LIN {X 0,Y 432.358,Z 386.63,A -85,B 0,C 180,E1 -9401.61,E2 -9401.61} C_VEL
LIN {X 0,Y 432.364,Z 386.63,A -85,B 0,C 180,E1 -9404.344,E2 -9404.344} C_VEL
LIN {X 0,Y 432.353,Z 386.63,A -85,B 0,C 180,E1 -9407.012,E2 -9407.012} C_VEL
LIN {X 0,Y 432.346,Z 386.632,A -85,B 0,C 180,E1 -9409.819,E2 -9409.819} C_VEL
LIN {X 0,Y 432.307,Z 386.637,A -85,B 0,C 180,E1 -9413.026,E2 -9413.026} C_VEL
LIN {X 0,Y 432.344,Z 386.755,A -85,B 0,C 180,E1 -9413.32,E2 -9413.32} C_VEL
LIN {X 0,Y 433.977,Z 394.809,A -85,B 0,C 180,E1 -9416.595,E2 -9416.595} C_VEL
LIN {X 0,Y 435.011,Z 400.873,A -85,B 0,C 180,E1 -9418.9,E2 -9418.9} C_VEL
LIN {X 0,Y 434.635,Z 406.92,A -85,B 0,C 180,E1 -9420.984,E2 -9420.984} C_VEL
LIN {X 0,Y 433.713,Z 417.772,A -85,B 0,C 180,E1 -9424.573,E2 -9424.573} C_VEL
LIN {X 0,Y 432.959,Z 428.81,A -85,B 0,C 180,E1 -9428.081,E2 -9428.081} C_VEL
LIN {X 0,Y 432.347,Z 440.008,A -85,B 0,C 180,E1 -9431.522,E2 -9431.522} C_VEL
LIN {X 0,Y 432.076,Z 446.933,A -85,B 0,C 180,E1 -9433.599,E2 -9433.599} C_VEL
LIN {X 0,Y 434.037,Z 460.55,A -85,B 0,C 180,E1 -9434.04,E2 -9434.04} C_VEL
LIN {X 0,Y 435.084,Z 471.816,A -85,B 0,C 180,E1 -9434.545,E2 -9434.545} C_VEL
LIN {X 0,Y 434.478,Z 484.277,A -85,B 0,C 180,E1 -9435.243,E2 -9435.243} C_VEL
LIN {X 0,Y 433.851,Z 495.5,A -85,B 0,C 180,E1 -9436.066,E2 -9436.066} C_VEL
LIN {X 0,Y 433.278,Z 505.592,A -85,B 0,C 180,E1 -9436.996,E2 -9436.996} C_VEL
LIN {X 0,Y 432.825,Z 514.915,A -85,B 0,C 180,E1 -9438.054,E2 -9438.054} C_VEL
LIN {X 0,Y 432.276,Z 523.539,A -85,B 0,C 180,E1 -9439.226,E2 -9439.226} C_VEL
LIN {X 0,Y 431.847,Z 531.941,A -85,B 0,C 180,E1 -9440.636,E2 -9440.636} C_VEL
LIN {X 0,Y 431.545,Z 538.678,A -85,B 0,C 180,E1 -9442.045,E2 -9442.045} C_VEL
LIN {X 0,Y 431.34,Z 544.033,A -85,B 0,C 180,E1 -9443.453,E2 -9443.453} C_VEL
LIN {X 0,Y 431.31,Z 548.179,A -85,B 0,C 180,E1 -9444.86,E2 -9444.86} C_VEL
LIN {X 0,Y 431.221,Z 551.229,A -85,B 0,C 180,E1 -9446.264,E2 -9446.264} C_VEL
LIN {X 0,Y 431.268,Z 552.713,A -85,B 0,C 180,E1 -9447.2,E2 -9447.2} C_VEL
LIN {X 0,Y 431.273,Z 553.741,A -85,B 0,C 180,E1 -9448.134,E2 -9448.134} C_VEL
LIN {X 0,Y 431.222,Z 554.368,A -85,B 0,C 180,E1 -9449.068,E2 -9449.068} C_VEL
LIN {X 0,Y 431.193,Z 554.599,A -85,B 0,C 180,E1 -9450.002,E2 -9450.002} C_VEL
LIN {X 0,Y 431.223,Z 554.385,A -85,B 0,C 180,E1 -9450.936,E2 -9450.936} C_VEL
LIN {X 0,Y 431.285,Z 553.758,A -85,B 0,C 180,E1 -9451.87,E2 -9451.87} C_VEL
LIN {X 0,Y 431.269,Z 552.732,A -85,B 0,C 180,E1 -9452.804,E2 -9452.804} C_VEL
LIN {X 0,Y 431.223,Z 551.283,A -85,B 0,C 180,E1 -9453.74,E2 -9453.74} C_VEL
LIN {X 0,Y 431.313,Z 548.261,A -85,B 0,C 180,E1 -9455.144,E2 -9455.144} C_VEL
LIN {X 0,Y 431.379,Z 544.16,A -85,B 0,C 180,E1 -9456.55,E2 -9456.55} C_VEL
LIN {X 0,Y 431.599,Z 537.834,A -85,B 0,C 180,E1 -9458.193,E2 -9458.193} C_VEL
LIN {X 0,Y 431.932,Z 530.939,A -85,B 0,C 180,E1 -9459.602,E2 -9459.602} C_VEL
LIN {X 0,Y 432.371,Z 522.327,A -85,B 0,C 180,E1 -9461.012,E2 -9461.012} C_VEL
LIN {X 0,Y 432.952,Z 513.464,A -85,B 0,C 180,E1 -9462.184,E2 -9462.184} C_VEL
LIN {X 0,Y 433.444,Z 503.391,A -85,B 0,C 180,E1 -9463.278,E2 -9463.278} C_VEL
LIN {X 0,Y 434.074,Z 493.107,A -85,B 0,C 180,E1 -9464.177,E2 -9464.177} C_VEL
LIN {X 0,Y 434.75,Z 481.287,A -85,B 0,C 180,E1 -9464.992,E2 -9464.992} C_VEL
LIN {X 0,Y 435.121,Z 470.397,A -85,B 0,C 180,E1 -9465.578,E2 -9465.578} C_VEL
LIN {X 0,Y 433.729,Z 457.18,A -85,B 0,C 180,E1 -9466.168,E2 -9466.168} C_VEL
LIN {X 0,Y 432.074,Z 446.577,A -85,B 0,C 180,E1 -9466.534,E2 -9466.534} C_VEL
LIN {X 0,Y 432.581,Z 435.274,A -85,B 0,C 180,E1 -9469.95,E2 -9469.95} C_VEL
LIN {X 0,Y 433.125,Z 425.632,A -85,B 0,C 180,E1 -9472.921,E2 -9472.921} C_VEL
LIN {X 0,Y 433.821,Z 416.066,A -85,B 0,C 180,E1 -9475.94,E2 -9475.94} C_VEL
LIN {X 0,Y 434.748,Z 404.887,A -85,B 0,C 180,E1 -9479.566,E2 -9479.566} C_VEL
LIN {X 0,Y 434.881,Z 400.204,A -85,B 0,C 180,E1 -9481.142,E2 -9481.142} C_VEL
LIN {X 0,Y 433.401,Z 391.79,A -85,B 0,C 180,E1 -9484.206,E2 -9484.206} C_VEL
LIN {X 0,Y 432.35,Z 386.632,A -85,B 0,C 180,E1 -9486.25,E2 -9486.25} C_VEL
LIN {X 0,Y 432.309,Z 386.636,A -85,B 0,C 180,E1 -9489.349,E2 -9489.349} C_VEL
LIN {X 0,Y 432.309,Z 386.637,A -85,B 0,C 180,E1 -9491.802,E2 -9491.802} C_VEL
LIN {X 0,Y 432.338,Z 386.63,A -85,B 0,C 180,E1 -9494.348,E2 -9494.348} C_VEL
LIN {X 0,Y 432.31,Z 386.633,A -85,B 0,C 180,E1 -9497.019,E2 -9497.019} C_VEL
LIN {X 0,Y 432.296,Z 386.633,A -85,B 0,C 180,E1 -9499.828,E2 -9499.828} C_VEL
LIN {X 0,Y 432.313,Z 386.634,A -85,B 0,C 180,E1 -9503.022,E2 -9503.022} C_VEL
LIN {X 0,Y 432.339,Z 386.632,A -85,B 0,C 180,E1 -9506.002,E2 -9506.002} C_VEL
LIN {X 0,Y 432.35,Z 386.631,A -85,B 0,C 180,E1 -9509.491,E2 -9509.491} C_VEL
LIN {X 0,Y 432.323,Z 386.634,A -85,B 0,C 180,E1 -9511.872,E2 -9511.872} C_VEL
LIN {X 0,Y 432.353,Z 386.629,A -85,B 0,C 180,E1 -9515.548,E2 -9515.548} C_VEL
LIN {X 0,Y 432.356,Z 386.63,A -85,B 0,C 180,E1 -9519.046,E2 -9519.046} C_VEL
LIN {X 0,Y 432.383,Z 386.628,A -85,B 0,C 180,E1 -9522.011,E2 -9522.011} C_VEL
LIN {X 0,Y 432.4,Z 386.625,A -85,B 0,C 180,E1 -9524.926,E2 -9524.926} C_VEL
LIN {X 0,Y 432.464,Z 386.618,A -85,B 0,C 180,E1 -9527.803,E2 -9527.803} C_VEL
LIN {X 0,Y 432.452,Z 386.619,A -85,B 0,C 180,E1 -9531.589,E2 -9531.589} C_VEL
LIN {X 0,Y 432.557,Z 386.607,A -85,B 0,C 180,E1 -9534.405,E2 -9534.405} C_VEL
LIN {X 0,Y 432.238,Z 386.721,A -85,B 0,C 180,E1 -9536.154,E2 -9536.154} C_VEL
LIN {X 0,Y 432.548,Z 392.214,A -85,B 0,C 180,E1 -9538.603,E2 -9538.603} C_VEL
LIN {X 0,Y 432.354,Z 397.392,A -85,B 0,C 180,E1 -9540.931,E2 -9540.931} C_VEL
LIN {X 0,Y 432.129,Z 406.596,A -85,B 0,C 180,E1 -9545.132,E2 -9545.132} C_VEL
LIN {X 0,Y 432.005,Z 412.681,A -85,B 0,C 180,E1 -9547.948,E2 -9547.948} C_VEL
LIN {X 0,Y 431.852,Z 419.741,A -85,B 0,C 180,E1 -9551.261,E2 -9551.261} C_VEL
LIN {X 0,Y 431.713,Z 426.157,A -85,B 0,C 180,E1 -9554.284,E2 -9554.284} C_VEL
LIN {X 0,Y 434.813,Z 440.469,A -85,B 0,C 180,E1 -9554.898,E2 -9554.898} C_VEL
LIN {X 0,Y 435.966,Z 447.264,A -85,B 0,C 180,E1 -9555.246,E2 -9555.246} C_VEL
LIN {X 0,Y 435.35,Z 459.685,A -85,B 0,C 180,E1 -9555.928,E2 -9555.928} C_VEL
LIN {X 0,Y 434.713,Z 471.741,A -85,B 0,C 180,E1 -9556.797,E2 -9556.797} C_VEL
LIN {X 0,Y 434.084,Z 482.032,A -85,B 0,C 180,E1 -9557.739,E2 -9557.739} C_VEL
LIN {X 0,Y 433.389,Z 492.493,A -85,B 0,C 180,E1 -9558.925,E2 -9558.925} C_VEL
LIN {X 0,Y 432.83,Z 501.477,A -85,B 0,C 180,E1 -9560.184,E2 -9560.184} C_VEL
LIN {X 0,Y 432.238,Z 510.153,A -85,B 0,C 180,E1 -9561.709,E2 -9561.709} C_VEL
LIN {X 0,Y 431.798,Z 517.081,A -85,B 0,C 180,E1 -9563.247,E2 -9563.247} C_VEL
LIN {X 0,Y 431.546,Z 521.85,A -85,B 0,C 180,E1 -9564.594,E2 -9564.594} C_VEL
LIN {X 0,Y 431.353,Z 526.477,A -85,B 0,C 180,E1 -9566.347,E2 -9566.347} C_VEL
LIN {X 0,Y 431.25,Z 528.08,A -85,B 0,C 180,E1 -9567.149,E2 -9567.149} C_VEL
LIN {X 0,Y 431.151,Z 529.853,A -85,B 0,C 180,E1 -9568.328,E2 -9568.328} C_VEL
LIN {X 0,Y 431.08,Z 530.807,A -85,B 0,C 180,E1 -9569.281,E2 -9569.281} C_VEL
LIN {X 0,Y 431.042,Z 531.392,A -85,B 0,C 180,E1 -9570.361,E2 -9570.361} C_VEL
LIN {X 0,Y 431.038,Z 531.205,A -85,B 0,C 180,E1 -9572.02,E2 -9572.02} C_VEL
LIN {X 0,Y 431.105,Z 529.669,A -85,B 0,C 180,E1 -9573.754,E2 -9573.754} C_VEL
LIN {X 0,Y 431.252,Z 526.839,A -85,B 0,C 180,E1 -9575.427,E2 -9575.427} C_VEL
LIN {X 0,Y 431.486,Z 522.666,A -85,B 0,C 180,E1 -9577.06,E2 -9577.06} C_VEL
LIN {X 0,Y 431.725,Z 517.333,A -85,B 0,C 180,E1 -9578.611,E2 -9578.611} C_VEL
LIN {X 0,Y 432.081,Z 510.568,A -85,B 0,C 180,E1 -9580.138,E2 -9580.138} C_VEL
LIN {X 0,Y 432.607,Z 502.081,A -85,B 0,C 180,E1 -9581.641,E2 -9581.641} C_VEL
LIN {X 0,Y 433.113,Z 494.004,A -85,B 0,C 180,E1 -9582.804,E2 -9582.804} C_VEL
LIN {X 0,Y 433.662,Z 485.008,A -85,B 0,C 180,E1 -9583.876,E2 -9583.876} C_VEL
LIN {X 0,Y 434.24,Z 474.608,A -85,B 0,C 180,E1 -9584.884,E2 -9584.884} C_VEL
LIN {X 0,Y 434.859,Z 463.18,A -85,B 0,C 180,E1 -9585.769,E2 -9585.769} C_VEL
LIN {X 0,Y 435.514,Z 450.906,A -85,B 0,C 180,E1 -9586.502,E2 -9586.502} C_VEL
LIN {X 0,Y 435.473,Z 445.507,A -85,B 0,C 180,E1 -9586.771,E2 -9586.771} C_VEL
LIN {X 0,Y 433.078,Z 432.684,A -85,B 0,C 180,E1 -9587.349,E2 -9587.349} C_VEL
LIN {X 0,Y 431.639,Z 425.615,A -85,B 0,C 180,E1 -9587.608,E2 -9587.608} C_VEL
LIN {X 0,Y 431.733,Z 419.417,A -85,B 0,C 180,E1 -9590.589,E2 -9590.589} C_VEL
LIN {X 0,Y 431.88,Z 412.017,A -85,B 0,C 180,E1 -9594.137,E2 -9594.137} C_VEL
LIN {X 0,Y 432.033,Z 406.117,A -85,B 0,C 180,E1 -9596.977,E2 -9596.977} C_VEL
LIN {X 0,Y 432.172,Z 399.276,A -85,B 0,C 180,E1 -9600.263,E2 -9600.263} C_VEL
LIN {X 0,Y 432.252,Z 392.712,A -85,B 0,C 180,E1 -9603.411,E2 -9603.411} C_VEL
LIN {X 0,Y 432.451,Z 386.619,A -85,B 0,C 180,E1 -9606.408,E2 -9606.408} C_VEL
LIN {X 0,Y 432.34,Z 386.632,A -85,B 0,C 180,E1 -9610.038,E2 -9610.038} C_VEL
LIN {X 0,Y 432.414,Z 386.624,A -85,B 0,C 180,E1 -9613.52,E2 -9613.52} C_VEL
LIN {X 0,Y 432.432,Z 386.62,A -85,B 0,C 180,E1 -9617.195,E2 -9617.195} C_VEL
LIN {X 0,Y 432.442,Z 386.618,A -85,B 0,C 180,E1 -9620.645,E2 -9620.645} C_VEL
LIN {X 0,Y 432.512,Z 386.61,A -85,B 0,C 180,E1 -9622.409,E2 -9622.409} C_VEL
LIN {X 0,Y 431.783,Z 386.704,A -85,B 0,C 180,E1 -9623.186,E2 -9623.186} C_VEL
LIN {X 0,Y 428.797,Z 387.08,A -85,B 0,C 180,E1 -9624.447,E2 -9624.447} C_VEL
LIN {X 0,Y 426.351,Z 387.384,A -85,B 0,C 180,E1 -9625.465,E2 -9625.465} C_VEL
LIN {X 0,Y 425.387,Z 387.502,A -85,B 0,C 180,E1 -9626.253,E2 -9626.253} C_VEL
LIN {X 0,Y 425.354,Z 387.503,A -85,B 0,C 180,E1 -9626.519,E2 -9626.519} C_VEL
LIN {X 0,Y 425.564,Z 387.52,A -85,B 0,C 180,E1 -9629.17,E2 -9629.17} C_VEL
LIN {X 0,Y 425.818,Z 388.833,A -85,B 0,C 180,E1 -9629.998,E2 -9629.998} C_VEL
LIN {X 0,Y 425.455,Z 393.602,A -85,B 0,C 180,E1 -9632.838,E2 -9632.838} C_VEL
LIN {X 0,Y 425.307,Z 398.421,A -85,B 0,C 180,E1 -9635.688,E2 -9635.688} C_VEL
LIN {X 0,Y 425.074,Z 403.376,A -85,B 0,C 180,E1 -9638.555,E2 -9638.555} C_VEL
LIN {X 0,Y 424.886,Z 410.151,A -85,B 0,C 180,E1 -9642.415,E2 -9642.415} C_VEL
LIN {X 0,Y 424.587,Z 417.168,A -85,B 0,C 180,E1 -9646.341,E2 -9646.341} C_VEL
LIN {X 0,Y 424.462,Z 422.693,A -85,B 0,C 180,E1 -9649.392,E2 -9649.392} C_VEL
LIN {X 0,Y 426.781,Z 435.095,A -85,B 0,C 180,E1 -9649.953,E2 -9649.953} C_VEL
LIN {X 0,Y 427.572,Z 441.78,A -85,B 0,C 180,E1 -9650.328,E2 -9650.328} C_VEL
LIN {X 0,Y 427.066,Z 453.282,A -85,B 0,C 180,E1 -9651.096,E2 -9651.096} C_VEL
LIN {X 0,Y 426.546,Z 462.376,A -85,B 0,C 180,E1 -9651.884,E2 -9651.884} C_VEL
LIN {X 0,Y 426.089,Z 471.591,A -85,B 0,C 180,E1 -9652.9,E2 -9652.9} C_VEL
LIN {X 0,Y 425.551,Z 480.362,A -85,B 0,C 180,E1 -9654.123,E2 -9654.123} C_VEL
LIN {X 0,Y 425.108,Z 487.845,A -85,B 0,C 180,E1 -9655.454,E2 -9655.454} C_VEL
LIN {X 0,Y 424.771,Z 493.266,A -85,B 0,C 180,E1 -9656.691,E2 -9656.691} C_VEL
LIN {X 0,Y 424.515,Z 498.155,A -85,B 0,C 180,E1 -9658.136,E2 -9658.136} C_VEL
LIN {X 0,Y 424.323,Z 502.024,A -85,B 0,C 180,E1 -9659.791,E2 -9659.791} C_VEL
LIN {X 0,Y 424.173,Z 503.721,A -85,B 0,C 180,E1 -9660.903,E2 -9660.903} C_VEL
LIN {X 0,Y 424.093,Z 504.894,A -85,B 0,C 180,E1 -9662.311,E2 -9662.311} C_VEL
LIN {X 0,Y 424.088,Z 505.08,A -85,B 0,C 180,E1 -9663.15,E2 -9663.15} C_VEL
LIN {X 0,Y 424.152,Z 504.719,A -85,B 0,C 180,E1 -9664.285,E2 -9664.285} C_VEL
LIN {X 0,Y 424.288,Z 503.202,A -85,B 0,C 180,E1 -9665.743,E2 -9665.743} C_VEL
LIN {X 0,Y 424.497,Z 500.104,A -85,B 0,C 180,E1 -9667.374,E2 -9667.374} C_VEL
LIN {X 0,Y 424.813,Z 495.456,A -85,B 0,C 180,E1 -9668.963,E2 -9668.963} C_VEL
LIN {X 0,Y 425.089,Z 490.857,A -85,B 0,C 180,E1 -9670.146,E2 -9670.146} C_VEL
LIN {X 0,Y 425.417,Z 484.917,A -85,B 0,C 180,E1 -9671.358,E2 -9671.358} C_VEL
LIN {X 0,Y 425.862,Z 477.403,A -85,B 0,C 180,E1 -9672.576,E2 -9672.576} C_VEL
LIN {X 0,Y 426.409,Z 469.473,A -85,B 0,C 180,E1 -9673.605,E2 -9673.605} C_VEL
LIN {X 0,Y 426.951,Z 460.386,A -85,B 0,C 180,E1 -9674.547,E2 -9674.547} C_VEL
LIN {X 0,Y 427.53,Z 450.085,A -85,B 0,C 180,E1 -9675.385,E2 -9675.385} C_VEL
LIN {X 0,Y 427.88,Z 440.687,A -85,B 0,C 180,E1 -9675.974,E2 -9675.974} C_VEL
LIN {X 0,Y 425.844,Z 429.204,A -85,B 0,C 180,E1 -9676.594,E2 -9676.594} C_VEL
LIN {X 0,Y 424.545,Z 423.172,A -85,B 0,C 180,E1 -9676.876,E2 -9676.876} C_VEL
LIN {X 0,Y 424.685,Z 416.884,A -85,B 0,C 180,E1 -9680.423,E2 -9680.423} C_VEL
LIN {X 0,Y 424.889,Z 410.362,A -85,B 0,C 180,E1 -9684.139,E2 -9684.139} C_VEL
LIN {X 0,Y 425.09,Z 404.684,A -85,B 0,C 180,E1 -9687.471,E2 -9687.471} C_VEL
LIN {X 0,Y 425.306,Z 399.882,A -85,B 0,C 180,E1 -9690.282,E2 -9690.282} C_VEL
LIN {X 0,Y 425.57,Z 394.467,A -85,B 0,C 180,E1 -9693.52,E2 -9693.52} C_VEL
LIN {X 0,Y 425.68,Z 391.017,A -85,B 0,C 180,E1 -9695.623,E2 -9695.623} C_VEL
LIN {X 0,Y 425.345,Z 387.506,A -85,B 0,C 180,E1 -9698.001,E2 -9698.001} C_VEL
LIN {X 0,Y 425.341,Z 387.508,A -85,B 0,C 180,E1 -9700.703,E2 -9700.703} C_VEL
LIN {X 0,Y 425.364,Z 387.505,A -85,B 0,C 180,E1 -9703.688,E2 -9703.688} C_VEL
LIN {X 0,Y 425.41,Z 387.496,A -85,B 0,C 180,E1 -9707.598,E2 -9707.598} C_VEL
LIN {X 0,Y 425.42,Z 387.495,A -85,B 0,C 180,E1 -9711.45,E2 -9711.45} C_VEL
LIN {X 0,Y 425.556,Z 387.478,A -85,B 0,C 180,E1 -9714.314,E2 -9714.314} C_VEL
LIN {X 0,Y 425.554,Z 387.476,A -85,B 0,C 180,E1 -9718.108,E2 -9718.108} C_VEL
LIN {X 0,Y 425.681,Z 387.461,A -85,B 0,C 180,E1 -9720,E2 -9720} C_VEL
LIN {X 0,Y 425.543,Z 387.479,A -85,B 0,C 180,E1 -9722.84,E2 -9722.84} C_VEL
LIN {X 0,Y 425.556,Z 387.478,A -85,B 0,C 180,E1 -9725.687,E2 -9725.687} C_VEL
LIN {X 0,Y 425.42,Z 387.495,A -85,B 0,C 180,E1 -9728.551,E2 -9728.551} C_VEL
LIN {X 0,Y 425.411,Z 387.493,A -85,B 0,C 180,E1 -9732.402,E2 -9732.402} C_VEL
LIN {X 0,Y 425.377,Z 387.497,A -85,B 0,C 180,E1 -9736.313,E2 -9736.313} C_VEL
LIN {X 0,Y 425.341,Z 387.505,A -85,B 0,C 180,E1 -9739.65,E2 -9739.65} C_VEL
LIN {X 0,Y 425.283,Z 387.511,A -85,B 0,C 180,E1 -9742.339,E2 -9742.339} C_VEL
LIN {X 0,Y 425.275,Z 387.511,A -85,B 0,C 180,E1 -9745.447,E2 -9745.447} C_VEL
LIN {X 0,Y 425.318,Z 387.508,A -85,B 0,C 180,E1 -9748.633,E2 -9748.633} C_VEL
LIN {X 0,Y 425.247,Z 387.512,A -85,B 0,C 180,E1 -9751.929,E2 -9751.929} C_VEL
LIN {X 0,Y 425.283,Z 387.512,A -85,B 0,C 180,E1 -9755.338,E2 -9755.338} C_VEL
LIN {X 0,Y 425.297,Z 387.51,A -85,B 0,C 180,E1 -9759.048,E2 -9759.048} C_VEL
LIN {X 0,Y 425.317,Z 387.507,A -85,B 0,C 180,E1 -9762.648,E2 -9762.648} C_VEL
LIN {X 0,Y 425.321,Z 387.508,A -85,B 0,C 180,E1 -9766.056,E2 -9766.056} C_VEL
LIN {X 0,Y 425.297,Z 387.509,A -85,B 0,C 180,E1 -9768.628,E2 -9768.628} C_VEL
LIN {X 0,Y 425.313,Z 387.508,A -85,B 0,C 180,E1 -9771.107,E2 -9771.107} C_VEL
LIN {X 0,Y 425.294,Z 387.61,A -85,B 0,C 180,E1 -9772.907,E2 -9772.907} C_VEL
LIN {X 0,Y 426.79,Z 394.85,A -85,B 0,C 180,E1 -9775.956,E2 -9775.956} C_VEL
LIN {X 0,Y 427.974,Z 401.737,A -85,B 0,C 180,E1 -9778.641,E2 -9778.641} C_VEL
LIN {X 0,Y 427.951,Z 405.329,A -85,B 0,C 180,E1 -9779.945,E2 -9779.945} C_VEL
LIN {X 0,Y 427.036,Z 414.755,A -85,B 0,C 180,E1 -9783.144,E2 -9783.144} C_VEL
LIN {X 0,Y 426.317,Z 423.905,A -85,B 0,C 180,E1 -9786.181,E2 -9786.181} C_VEL
LIN {X 0,Y 425.606,Z 435.019,A -85,B 0,C 180,E1 -9789.713,E2 -9789.713} C_VEL
LIN {X 0,Y 425.052,Z 446.04,A -85,B 0,C 180,E1 -9793.134,E2 -9793.134} C_VEL
LIN {X 0,Y 425.03,Z 446.677,A -85,B 0,C 180,E1 -9793.328,E2 -9793.328} C_VEL
LIN {X 0,Y 427.067,Z 460.804,A -85,B 0,C 180,E1 -9793.803,E2 -9793.803} C_VEL
LIN {X 0,Y 428.185,Z 472.48,A -85,B 0,C 180,E1 -9794.35,E2 -9794.35} C_VEL
LIN {X 0,Y 427.587,Z 483.807,A -85,B 0,C 180,E1 -9794.999,E2 -9794.999} C_VEL
LIN {X 0,Y 426.919,Z 495.116,A -85,B 0,C 180,E1 -9795.84,E2 -9795.84} C_VEL
LIN {X 0,Y 426.331,Z 504.628,A -85,B 0,C 180,E1 -9796.725,E2 -9796.725} C_VEL
LIN {X 0,Y 425.826,Z 514.507,A -85,B 0,C 180,E1 -9797.855,E2 -9797.855} C_VEL
LIN {X 0,Y 425.25,Z 523.184,A -85,B 0,C 180,E1 -9799.046,E2 -9799.046} C_VEL
LIN {X 0,Y 424.793,Z 531.626,A -85,B 0,C 180,E1 -9800.479,E2 -9800.479} C_VEL
LIN {X 0,Y 424.496,Z 538.388,A -85,B 0,C 180,E1 -9801.912,E2 -9801.912} C_VEL
LIN {X 0,Y 424.255,Z 543.764,A -85,B 0,C 180,E1 -9803.343,E2 -9803.343} C_VEL
LIN {X 0,Y 424.221,Z 547.93,A -85,B 0,C 180,E1 -9804.774,E2 -9804.774} C_VEL
LIN {X 0,Y 424.13,Z 550.997,A -85,B 0,C 180,E1 -9806.202,E2 -9806.202} C_VEL
LIN {X 0,Y 424.164,Z 552.497,A -85,B 0,C 180,E1 -9807.153,E2 -9807.153} C_VEL
LIN {X 0,Y 424.194,Z 553.533,A -85,B 0,C 180,E1 -9808.103,E2 -9808.103} C_VEL
LIN {X 0,Y 424.139,Z 554.167,A -85,B 0,C 180,E1 -9809.053,E2 -9809.053} C_VEL
LIN {X 0,Y 424.109,Z 554.405,A -85,B 0,C 180,E1 -9810.002,E2 -9810.002} C_VEL
LIN {X 0,Y 424.141,Z 554.202,A -85,B 0,C 180,E1 -9810.952,E2 -9810.952} C_VEL
LIN {X 0,Y 424.205,Z 553.581,A -85,B 0,C 180,E1 -9811.901,E2 -9811.901} C_VEL
LIN {X 0,Y 424.165,Z 552.557,A -85,B 0,C 180,E1 -9812.851,E2 -9812.851} C_VEL
LIN {X 0,Y 424.132,Z 551.117,A -85,B 0,C 180,E1 -9813.802,E2 -9813.802} C_VEL
LIN {X 0,Y 424.225,Z 548.103,A -85,B 0,C 180,E1 -9815.23,E2 -9815.23} C_VEL
LIN {X 0,Y 424.302,Z 544.011,A -85,B 0,C 180,E1 -9816.66,E2 -9816.66} C_VEL
LIN {X 0,Y 424.53,Z 537.692,A -85,B 0,C 180,E1 -9818.331,E2 -9818.331} C_VEL
LIN {X 0,Y 424.88,Z 530.806,A -85,B 0,C 180,E1 -9819.763,E2 -9819.763} C_VEL
LIN {X 0,Y 425.286,Z 523.782,A -85,B 0,C 180,E1 -9820.957,E2 -9820.957} C_VEL
LIN {X 0,Y 425.855,Z 515.334,A -85,B 0,C 180,E1 -9822.149,E2 -9822.149} C_VEL
LIN {X 0,Y 426.421,Z 504.9,A -85,B 0,C 180,E1 -9823.342,E2 -9823.342} C_VEL
LIN {X 0,Y 427.191,Z 493.2,A -85,B 0,C 180,E1 -9824.41,E2 -9824.41} C_VEL
LIN {X 0,Y 427.913,Z 481.485,A -85,B 0,C 180,E1 -9825.237,E2 -9825.237} C_VEL
LIN {X 0,Y 428.232,Z 470.736,A -85,B 0,C 180,E1 -9825.835,E2 -9825.835} C_VEL
LIN {X 0,Y 426.877,Z 457.574,A -85,B 0,C 180,E1 -9826.444,E2 -9826.444} C_VEL
LIN {X 0,Y 425.037,Z 446.206,A -85,B 0,C 180,E1 -9826.84,E2 -9826.84} C_VEL
LIN {X 0,Y 425.584,Z 434.989,A -85,B 0,C 180,E1 -9830.293,E2 -9830.293} C_VEL
LIN {X 0,Y 426.171,Z 425.419,A -85,B 0,C 180,E1 -9833.317,E2 -9833.317} C_VEL
LIN {X 0,Y 426.896,Z 415.862,A -85,B 0,C 180,E1 -9836.393,E2 -9836.393} C_VEL
LIN {X 0,Y 427.755,Z 406.371,A -85,B 0,C 180,E1 -9839.533,E2 -9839.533} C_VEL
LIN {X 0,Y 427.958,Z 402.187,A -85,B 0,C 180,E1 -9840.962,E2 -9840.962} C_VEL
LIN {X 0,Y 426.844,Z 395.332,A -85,B 0,C 180,E1 -9843.476,E2 -9843.476} C_VEL
LIN {X 0,Y 425.286,Z 387.512,A -85,B 0,C 180,E1 -9846.508,E2 -9846.508} C_VEL
LIN {X 0,Y 425.269,Z 387.513,A -85,B 0,C 180,E1 -9849.038,E2 -9849.038} C_VEL
LIN {X 0,Y 425.261,Z 387.512,A -85,B 0,C 180,E1 -9852.656,E2 -9852.656} C_VEL
LIN {X 0,Y 425.29,Z 387.511,A -85,B 0,C 180,E1 -9855.284,E2 -9855.284} C_VEL
LIN {X 0,Y 425.255,Z 387.512,A -85,B 0,C 180,E1 -9858.619,E2 -9858.619} C_VEL
LIN {X 0,Y 425.288,Z 387.507,A -85,B 0,C 180,E1 -9861.1,E2 -9861.1} C_VEL
LIN {X 0,Y 425.302,Z 387.509,A -85,B 0,C 180,E1 -9864.664,E2 -9864.664} C_VEL
LIN {X 0,Y 425.269,Z 387.514,A -85,B 0,C 180,E1 -9868.073,E2 -9868.073} C_VEL
LIN {X 0,Y 425.302,Z 387.511,A -85,B 0,C 180,E1 -9871.365,E2 -9871.365} C_VEL
LIN {X 0,Y 425.256,Z 387.513,A -85,B 0,C 180,E1 -9874.552,E2 -9874.552} C_VEL
LIN {X 0,Y 425.298,Z 387.507,A -85,B 0,C 180,E1 -9877.73,E2 -9877.73} C_VEL
LIN {X 0,Y 425.368,Z 387.501,A -85,B 0,C 180,E1 -9880.704,E2 -9880.704} C_VEL
LIN {X 0,Y 425.395,Z 387.499,A -85,B 0,C 180,E1 -9883.688,E2 -9883.688} C_VEL
LIN {X 0,Y 425.417,Z 387.496,A -85,B 0,C 180,E1 -9887.598,E2 -9887.598} C_VEL
LIN {X 0,Y 425.4,Z 387.498,A -85,B 0,C 180,E1 -9891.449,E2 -9891.449} C_VEL
LIN {X 0,Y 425.514,Z 387.484,A -85,B 0,C 180,E1 -9894.312,E2 -9894.312} C_VEL
LIN {X 0,Y 425.246,Z 387.608,A -85,B 0,C 180,E1 -9895.972,E2 -9895.972} C_VEL
LIN {X 0,Y 425.548,Z 393.357,A -85,B 0,C 180,E1 -9898.58,E2 -9898.58} C_VEL
LIN {X 0,Y 425.298,Z 399.705,A -85,B 0,C 180,E1 -9901.42,E2 -9901.42} C_VEL
LIN {X 0,Y 425.11,Z 407.729,A -85,B 0,C 180,E1 -9905.217,E2 -9905.217} C_VEL
LIN {X 0,Y 424.975,Z 413.93,A -85,B 0,C 180,E1 -9908.08,E2 -9908.08} C_VEL
LIN {X 0,Y 424.801,Z 421.048,A -85,B 0,C 180,E1 -9911.451,E2 -9911.451} C_VEL
LIN {X 0,Y 424.659,Z 426.363,A -85,B 0,C 180,E1 -9913.976,E2 -9913.976} C_VEL
LIN {X 0,Y 427.746,Z 440.102,A -85,B 0,C 180,E1 -9914.571,E2 -9914.571} C_VEL
LIN {X 0,Y 429.138,Z 448.31,A -85,B 0,C 180,E1 -9915.008,E2 -9915.008} C_VEL
LIN {X 0,Y 428.525,Z 460.474,A -85,B 0,C 180,E1 -9915.7,E2 -9915.7} C_VEL
LIN {X 0,Y 427.845,Z 472.367,A -85,B 0,C 180,E1 -9916.583,E2 -9916.583} C_VEL
LIN {X 0,Y 427.183,Z 482.324,A -85,B 0,C 180,E1 -9917.515,E2 -9917.515} C_VEL
LIN {X 0,Y 426.444,Z 492.98,A -85,B 0,C 180,E1 -9918.745,E2 -9918.745} C_VEL
LIN {X 0,Y 425.857,Z 501.672,A -85,B 0,C 180,E1 -9919.987,E2 -9919.987} C_VEL
LIN {X 0,Y 425.233,Z 510.338,A -85,B 0,C 180,E1 -9921.535,E2 -9921.535} C_VEL
LIN {X 0,Y 424.852,Z 516.372,A -85,B 0,C 180,E1 -9922.876,E2 -9922.876} C_VEL
LIN {X 0,Y 424.489,Z 521.996,A -85,B 0,C 180,E1 -9924.45,E2 -9924.45} C_VEL
LIN {X 0,Y 424.286,Z 526.182,A -85,B 0,C 180,E1 -9926.023,E2 -9926.023} C_VEL
LIN {X 0,Y 424.1,Z 529.214,A -85,B 0,C 180,E1 -9927.645,E2 -9927.645} C_VEL
LIN {X 0,Y 424.032,Z 530.579,A -85,B 0,C 180,E1 -9928.728,E2 -9928.728} C_VEL
LIN {X 0,Y 423.94,Z 531.603,A -85,B 0,C 180,E1 -9930.451,E2 -9930.451} C_VEL
LIN {X 0,Y 423.953,Z 531.26,A -85,B 0,C 180,E1 -9932.279,E2 -9932.279} C_VEL
LIN {X 0,Y 424.038,Z 529.534,A -85,B 0,C 180,E1 -9934.033,E2 -9934.033} C_VEL
LIN {X 0,Y 424.211,Z 526.476,A -85,B 0,C 180,E1 -9935.727,E2 -9935.727} C_VEL
LIN {X 0,Y 424.453,Z 522.18,A -85,B 0,C 180,E1 -9937.365,E2 -9937.365} C_VEL
LIN {X 0,Y 424.695,Z 516.553,A -85,B 0,C 180,E1 -9938.964,E2 -9938.964} C_VEL
LIN {X 0,Y 425.145,Z 509.565,A -85,B 0,C 180,E1 -9940.497,E2 -9940.497} C_VEL
LIN {X 0,Y 425.615,Z 501.931,A -85,B 0,C 180,E1 -9941.847,E2 -9941.847} C_VEL
LIN {X 0,Y 426.149,Z 493.785,A -85,B 0,C 180,E1 -9943.027,E2 -9943.027} C_VEL
LIN {X 0,Y 426.805,Z 483.418,A -85,B 0,C 180,E1 -9944.248,E2 -9944.248} C_VEL
LIN {X 0,Y 427.48,Z 472.07,A -85,B 0,C 180,E1 -9945.32,E2 -9945.32} C_VEL
LIN {X 0,Y 428.09,Z 460.713,A -85,B 0,C 180,E1 -9946.164,E2 -9946.164} C_VEL
LIN {X 0,Y 428.761,Z 447.732,A -85,B 0,C 180,E1 -9946.896,E2 -9946.896} C_VEL
LIN {X 0,Y 426.433,Z 434.83,A -85,B 0,C 180,E1 -9947.519,E2 -9947.519} C_VEL
LIN {X 0,Y 424.555,Z 425.773,A -85,B 0,C 180,E1 -9947.858,E2 -9947.858} C_VEL
LIN {X 0,Y 424.684,Z 419.162,A -85,B 0,C 180,E1 -9951.058,E2 -9951.058} C_VEL
LIN {X 0,Y 424.831,Z 412.763,A -85,B 0,C 180,E1 -9954.155,E2 -9954.155} C_VEL
LIN {X 0,Y 424.978,Z 407.052,A -85,B 0,C 180,E1 -9956.924,E2 -9956.924} C_VEL
LIN {X 0,Y 425.131,Z 400.159,A -85,B 0,C 180,E1 -9960.267,E2 -9960.267} C_VEL
LIN {X 0,Y 425.225,Z 393.502,A -85,B 0,C 180,E1 -9963.495,E2 -9963.495} C_VEL
LIN {X 0,Y 425.419,Z 387.495,A -85,B 0,C 180,E1 -9966.446,E2 -9966.446} C_VEL
LIN {X 0,Y 425.33,Z 387.508,A -85,B 0,C 180,E1 -9970.363,E2 -9970.363} C_VEL
LIN {X 0,Y 425.39,Z 387.5,A -85,B 0,C 180,E1 -9973.687,E2 -9973.687} C_VEL
LIN {X 0,Y 425.413,Z 387.493,A -85,B 0,C 180,E1 -9977.596,E2 -9977.596} C_VEL
LIN {X 0,Y 425.437,Z 387.494,A -85,B 0,C 180,E1 -9981.448,E2 -9981.448} C_VEL
LIN {X 0,Y 425.539,Z 387.482,A -85,B 0,C 180,E1 -9984.311,E2 -9984.311} C_VEL
LIN {X 0,Y 425.354,Z 387.503,A -85,B 0,C 180,E1 -9986.519,E2 -9986.519} C_VEL
LIN {X 0,Y 424.849,Z 387.617,A -85,B 0,C 180,E1 -9987.309,E2 -9987.309} C_VEL
LIN {X 0,Y 422.195,Z 388.377,A -85,B 0,C 180,E1 -9988.593,E2 -9988.593} C_VEL
LIN {X 0,Y 419.851,Z 389.477,A -85,B 0,C 180,E1 -9989.622,E2 -9989.622} C_VEL
LIN {X 0,Y 418.804,Z 390.583,A -85,B 0,C 180,E1 -9990.41,E2 -9990.41} C_VEL
LIN {X 0,Y 418.702,Z 391.004,A -85,B 0,C 180,E1 -9990.675,E2 -9990.675} C_VEL
LIN {X 0,Y 418.234,Z 396.293,A -85,B 0,C 180,E1 -9993.852,E2 -9993.852} C_VEL
LIN {X 0,Y 418.168,Z 401.178,A -85,B 0,C 180,E1 -9996.754,E2 -9996.754} C_VEL
LIN {X 0,Y 417.94,Z 406.195,A -85,B 0,C 180,E1 -9999.678,E2 -9999.678} C_VEL
LIN {X 0,Y 417.809,Z 411.399,A -85,B 0,C 180,E1 -10002.679,E2 -10002.679} C_VEL
LIN {X 0,Y 417.502,Z 418.387,A -85,B 0,C 180,E1 -10006.626,E2 -10006.626} C_VEL
LIN {X 0,Y 417.378,Z 422.882,A -85,B 0,C 180,E1 -10009.147,E2 -10009.147} C_VEL
LIN {X 0,Y 419.661,Z 434.815,A -85,B 0,C 180,E1 -10009.691,E2 -10009.691} C_VEL
LIN {X 0,Y 420.669,Z 442.52,A -85,B 0,C 180,E1 -10010.135,E2 -10010.135} C_VEL
LIN {X 0,Y 420.149,Z 453.656,A -85,B 0,C 180,E1 -10010.897,E2 -10010.897} C_VEL
LIN {X 0,Y 419.573,Z 463.243,A -85,B 0,C 180,E1 -10011.75,E2 -10011.75} C_VEL
LIN {X 0,Y 419.104,Z 471.998,A -85,B 0,C 180,E1 -10012.736,E2 -10012.736} C_VEL
LIN {X 0,Y 418.65,Z 479.358,A -85,B 0,C 180,E1 -10013.756,E2 -10013.756} C_VEL
LIN {X 0,Y 418.151,Z 486.97,A -85,B 0,C 180,E1 -10015.082,E2 -10015.082} C_VEL
LIN {X 0,Y 417.786,Z 492.973,A -85,B 0,C 180,E1 -10016.41,E2 -10016.41} C_VEL
LIN {X 0,Y 417.558,Z 497.08,A -85,B 0,C 180,E1 -10017.568,E2 -10017.568} C_VEL
LIN {X 0,Y 417.351,Z 501.418,A -85,B 0,C 180,E1 -10019.229,E2 -10019.229} C_VEL
LIN {X 0,Y 417.125,Z 503.988,A -85,B 0,C 180,E1 -10020.765,E2 -10020.765} C_VEL
LIN {X 0,Y 417.047,Z 504.757,A -85,B 0,C 180,E1 -10021.49,E2 -10021.49} C_VEL
LIN {X 0,Y 417.022,Z 505.407,A -85,B 0,C 180,E1 -10022.632,E2 -10022.632} C_VEL
LIN {X 0,Y 417.085,Z 505.11,A -85,B 0,C 180,E1 -10024.345,E2 -10024.345} C_VEL
LIN {X 0,Y 417.244,Z 503.141,A -85,B 0,C 180,E1 -10026.12,E2 -10026.12} C_VEL
LIN {X 0,Y 417.464,Z 499.92,A -85,B 0,C 180,E1 -10027.699,E2 -10027.699} C_VEL
LIN {X 0,Y 417.837,Z 495.063,A -85,B 0,C 180,E1 -10029.312,E2 -10029.312} C_VEL
LIN {X 0,Y 418.237,Z 488.595,A -85,B 0,C 180,E1 -10030.873,E2 -10030.873} C_VEL
LIN {X 0,Y 418.67,Z 481.527,A -85,B 0,C 180,E1 -10032.176,E2 -10032.176} C_VEL
LIN {X 0,Y 419.235,Z 473.029,A -85,B 0,C 180,E1 -10033.414,E2 -10033.414} C_VEL
LIN {X 0,Y 419.91,Z 463.137,A -85,B 0,C 180,E1 -10034.538,E2 -10034.538} C_VEL
LIN {X 0,Y 420.525,Z 452.656,A -85,B 0,C 180,E1 -10035.456,E2 -10035.456} C_VEL
LIN {X 0,Y 421.018,Z 441.963,A -85,B 0,C 180,E1 -10036.169,E2 -10036.169} C_VEL
LIN {X 0,Y 418.939,Z 430.236,A -85,B 0,C 180,E1 -10036.833,E2 -10036.833} C_VEL
LIN {X 0,Y 417.512,Z 423.439,A -85,B 0,C 180,E1 -10037.144,E2 -10037.144} C_VEL
LIN {X 0,Y 417.657,Z 417.183,A -85,B 0,C 180,E1 -10040.714,E2 -10040.714} C_VEL
LIN {X 0,Y 417.869,Z 410.597,A -85,B 0,C 180,E1 -10044.533,E2 -10044.533} C_VEL
LIN {X 0,Y 418.059,Z 405.653,A -85,B 0,C 180,E1 -10047.456,E2 -10047.456} C_VEL
LIN {X 0,Y 418.324,Z 399.975,A -85,B 0,C 180,E1 -10050.875,E2 -10050.875} C_VEL
LIN {X 0,Y 418.565,Z 394.644,A -85,B 0,C 180,E1 -10054.116,E2 -10054.116} C_VEL
LIN {X 0,Y 418.603,Z 391.231,A -85,B 0,C 180,E1 -10056.238,E2 -10056.238} C_VEL
LIN {X 0,Y 418.308,Z 388.383,A -85,B 0,C 180,E1 -10058.198,E2 -10058.198} C_VEL
LIN {X 0,Y 418.261,Z 388.39,A -85,B 0,C 180,E1 -10061.382,E2 -10061.382} C_VEL
LIN {X 0,Y 418.28,Z 388.387,A -85,B 0,C 180,E1 -10064.405,E2 -10064.405} C_VEL
LIN {X 0,Y 418.349,Z 388.376,A -85,B 0,C 180,E1 -10067.386,E2 -10067.386} C_VEL
LIN {X 0,Y 418.34,Z 388.377,A -85,B 0,C 180,E1 -10070.329,E2 -10070.329} C_VEL
LIN {X 0,Y 418.472,Z 388.36,A -85,B 0,C 180,E1 -10073.249,E2 -10073.249} C_VEL
LIN {X 0,Y 418.326,Z 388.38,A -85,B 0,C 180,E1 -10075.182,E2 -10075.182} C_VEL
LIN {X 0,Y 418.523,Z 388.352,A -85,B 0,C 180,E1 -10078.076,E2 -10078.076} C_VEL
LIN {X 0,Y 418.651,Z 388.337,A -85,B 0,C 180,E1 -10080,E2 -10080} C_VEL
LIN {X 0,Y 418.497,Z 388.357,A -85,B 0,C 180,E1 -10082.888,E2 -10082.888} C_VEL
LIN {X 0,Y 418.511,Z 388.356,A -85,B 0,C 180,E1 -10085.783,E2 -10085.783} C_VEL
LIN {X 0,Y 418.378,Z 388.371,A -85,B 0,C 180,E1 -10088.696,E2 -10088.696} C_VEL
LIN {X 0,Y 418.318,Z 388.378,A -85,B 0,C 180,E1 -10091.631,E2 -10091.631} C_VEL
LIN {X 0,Y 418.291,Z 388.381,A -85,B 0,C 180,E1 -10094.598,E2 -10094.598} C_VEL
LIN {X 0,Y 418.269,Z 388.385,A -85,B 0,C 180,E1 -10097.605,E2 -10097.605} C_VEL
LIN {X 0,Y 418.255,Z 388.386,A -85,B 0,C 180,E1 -10100.663,E2 -10100.663} C_VEL
LIN {X 0,Y 418.271,Z 388.382,A -85,B 0,C 180,E1 -10103.782,E2 -10103.782} C_VEL
LIN {X 0,Y 418.29,Z 388.379,A -85,B 0,C 180,E1 -10107.072,E2 -10107.072} C_VEL
LIN {X 0,Y 418.241,Z 388.387,A -85,B 0,C 180,E1 -10110.273,E2 -10110.273} C_VEL
LIN {X 0,Y 418.23,Z 388.389,A -85,B 0,C 180,E1 -10113.679,E2 -10113.679} C_VEL
LIN {X 0,Y 418.23,Z 388.389,A -85,B 0,C 180,E1 -10117.226,E2 -10117.226} C_VEL
LIN {X 0,Y 418.25,Z 388.388,A -85,B 0,C 180,E1 -10119.682,E2 -10119.682} C_VEL
LIN {X 0,Y 418.27,Z 388.386,A -85,B 0,C 180,E1 -10122.332,E2 -10122.332} C_VEL
LIN {X 0,Y 418.26,Z 388.384,A -85,B 0,C 180,E1 -10125.116,E2 -10125.116} C_VEL
LIN {X 0,Y 418.28,Z 388.385,A -85,B 0,C 180,E1 -10127.776,E2 -10127.776} C_VEL
LIN {X 0,Y 418.256,Z 388.389,A -85,B 0,C 180,E1 -10131.562,E2 -10131.562} C_VEL
LIN {X 0,Y 418.248,Z 388.437,A -85,B 0,C 180,E1 -10132.476,E2 -10132.476} C_VEL
LIN {X 0,Y 419.891,Z 396.393,A -85,B 0,C 180,E1 -10135.899,E2 -10135.899} C_VEL
LIN {X 0,Y 420.953,Z 402.563,A -85,B 0,C 180,E1 -10138.372,E2 -10138.372} C_VEL
LIN {X 0,Y 420.982,Z 406.835,A -85,B 0,C 180,E1 -10139.948,E2 -10139.948} C_VEL
LIN {X 0,Y 420.019,Z 416.034,A -85,B 0,C 180,E1 -10143.145,E2 -10143.145} C_VEL
LIN {X 0,Y 419.264,Z 425.351,A -85,B 0,C 180,E1 -10146.281,E2 -10146.281} C_VEL
LIN {X 0,Y 418.613,Z 434.803,A -85,B 0,C 180,E1 -10149.359,E2 -10149.359} C_VEL
LIN {X 0,Y 418.02,Z 445.759,A -85,B 0,C 180,E1 -10152.841,E2 -10152.841} C_VEL
LIN {X 0,Y 417.983,Z 446.422,A -85,B 0,C 180,E1 -10153.048,E2 -10153.048} C_VEL
LIN {X 0,Y 420.103,Z 460.623,A -85,B 0,C 180,E1 -10153.543,E2 -10153.543} C_VEL
LIN {X 0,Y 421.28,Z 473.108,A -85,B 0,C 180,E1 -10154.15,E2 -10154.15} C_VEL
LIN {X 0,Y 420.614,Z 485.116,A -85,B 0,C 180,E1 -10154.869,E2 -10154.869} C_VEL
LIN {X 0,Y 419.895,Z 496.247,A -85,B 0,C 180,E1 -10155.734,E2 -10155.734} C_VEL
LIN {X 0,Y 419.239,Z 506.819,A -85,B 0,C 180,E1 -10156.782,E2 -10156.782} C_VEL
LIN {X 0,Y 418.599,Z 517.783,A -85,B 0,C 180,E1 -10158.134,E2 -10158.134} C_VEL
LIN {X 0,Y 418.021,Z 525.859,A -85,B 0,C 180,E1 -10159.345,E2 -10159.345} C_VEL
LIN {X 0,Y 417.618,Z 533.766,A -85,B 0,C 180,E1 -10160.803,E2 -10160.803} C_VEL
LIN {X 0,Y 417.33,Z 540.045,A -85,B 0,C 180,E1 -10162.26,E2 -10162.26} C_VEL
LIN {X 0,Y 417.097,Z 545.251,A -85,B 0,C 180,E1 -10163.795,E2 -10163.795} C_VEL
LIN {X 0,Y 417.119,Z 548.819,A -85,B 0,C 180,E1 -10165.17,E2 -10165.17} C_VEL
LIN {X 0,Y 417.043,Z 550.766,A -85,B 0,C 180,E1 -10166.137,E2 -10166.137} C_VEL
LIN {X 0,Y 417.061,Z 552.28,A -85,B 0,C 180,E1 -10167.104,E2 -10167.104} C_VEL
LIN {X 0,Y 417.117,Z 553.326,A -85,B 0,C 180,E1 -10168.071,E2 -10168.071} C_VEL
LIN {X 0,Y 417.059,Z 553.966,A -85,B 0,C 180,E1 -10169.037,E2 -10169.037} C_VEL
LIN {X 0,Y 417.028,Z 554.21,A -85,B 0,C 180,E1 -10170.002,E2 -10170.002} C_VEL
LIN {X 0,Y 417.061,Z 554.019,A -85,B 0,C 180,E1 -10170.968,E2 -10170.968} C_VEL
LIN {X 0,Y 417.127,Z 553.402,A -85,B 0,C 180,E1 -10171.933,E2 -10171.933} C_VEL
LIN {X 0,Y 417.061,Z 552.382,A -85,B 0,C 180,E1 -10172.9,E2 -10172.9} C_VEL
LIN {X 0,Y 417.045,Z 550.951,A -85,B 0,C 180,E1 -10173.867,E2 -10173.867} C_VEL
LIN {X 0,Y 417.14,Z 547.943,A -85,B 0,C 180,E1 -10175.319,E2 -10175.319} C_VEL
LIN {X 0,Y 417.234,Z 543.863,A -85,B 0,C 180,E1 -10176.773,E2 -10176.773} C_VEL
LIN {X 0,Y 417.487,Z 537.569,A -85,B 0,C 180,E1 -10178.472,E2 -10178.472} C_VEL
LIN {X 0,Y 417.852,Z 530.713,A -85,B 0,C 180,E1 -10179.929,E2 -10179.929} C_VEL
LIN {X 0,Y 418.303,Z 523.726,A -85,B 0,C 180,E1 -10181.142,E2 -10181.142} C_VEL
LIN {X 0,Y 418.894,Z 515.311,A -85,B 0,C 180,E1 -10182.354,E2 -10182.354} C_VEL
LIN {X 0,Y 419.508,Z 504.924,A -85,B 0,C 180,E1 -10183.566,E2 -10183.566} C_VEL
LIN {X 0,Y 420.312,Z 493.286,A -85,B 0,C 180,E1 -10184.651,E2 -10184.651} C_VEL
LIN {X 0,Y 421.085,Z 481.683,A -85,B 0,C 180,E1 -10185.49,E2 -10185.49} C_VEL
LIN {X 0,Y 421.468,Z 472.311,A -85,B 0,C 180,E1 -10186.034,E2 -10186.034} C_VEL
LIN {X 0,Y 420.059,Z 457.937,A -85,B 0,C 180,E1 -10186.729,E2 -10186.729} C_VEL
LIN {X 0,Y 418.021,Z 445.705,A -85,B 0,C 180,E1 -10187.191,E2 -10187.191} C_VEL
LIN {X 0,Y 418.6,Z 434.739,A -85,B 0,C 180,E1 -10190.647,E2 -10190.647} C_VEL
LIN {X 0,Y 419.352,Z 423.561,A -85,B 0,C 180,E1 -10194.244,E2 -10194.244} C_VEL
LIN {X 0,Y 420.299,Z 412.501,A -85,B 0,C 180,E1 -10197.919,E2 -10197.919} C_VEL
LIN {X 0,Y 421.002,Z 404.624,A -85,B 0,C 180,E1 -10200.609,E2 -10200.609} C_VEL
LIN {X 0,Y 420.47,Z 399.883,A -85,B 0,C 180,E1 -10202.337,E2 -10202.337} C_VEL
LIN {X 0,Y 418.985,Z 392.055,A -85,B 0,C 180,E1 -10205.36,E2 -10205.36} C_VEL
LIN {X 0,Y 418.242,Z 388.389,A -85,B 0,C 180,E1 -10206.836,E2 -10206.836} C_VEL
LIN {X 0,Y 418.207,Z 388.394,A -85,B 0,C 180,E1 -10209.689,E2 -10209.689} C_VEL
LIN {X 0,Y 418.213,Z 388.392,A -85,B 0,C 180,E1 -10212.318,E2 -10212.318} C_VEL
LIN {X 0,Y 418.241,Z 388.389,A -85,B 0,C 180,E1 -10215.109,E2 -10215.109} C_VEL
LIN {X 0,Y 418.227,Z 388.388,A -85,B 0,C 180,E1 -10217.765,E2 -10217.765} C_VEL
LIN {X 0,Y 418.245,Z 388.382,A -85,B 0,C 180,E1 -10221.557,E2 -10221.557} C_VEL
LIN {X 0,Y 418.258,Z 388.384,A -85,B 0,C 180,E1 -10225.158,E2 -10225.158} C_VEL
LIN {X 0,Y 418.25,Z 388.386,A -85,B 0,C 180,E1 -10227.472,E2 -10227.472} C_VEL
LIN {X 0,Y 418.266,Z 388.383,A -85,B 0,C 180,E1 -10230.898,E2 -10230.898} C_VEL
LIN {X 0,Y 418.216,Z 388.389,A -85,B 0,C 180,E1 -10234.092,E2 -10234.092} C_VEL
LIN {X 0,Y 418.233,Z 388.389,A -85,B 0,C 180,E1 -10237.263,E2 -10237.263} C_VEL
LIN {X 0,Y 418.29,Z 388.383,A -85,B 0,C 180,E1 -10240.364,E2 -10240.364} C_VEL
LIN {X 0,Y 418.324,Z 388.378,A -85,B 0,C 180,E1 -10243.405,E2 -10243.405} C_VEL
LIN {X 0,Y 418.352,Z 388.375,A -85,B 0,C 180,E1 -10247,E2 -10247} C_VEL
LIN {X 0,Y 418.331,Z 388.376,A -85,B 0,C 180,E1 -10250.328,E2 -10250.328} C_VEL
LIN {X 0,Y 418.446,Z 388.366,A -85,B 0,C 180,E1 -10253.248,E2 -10253.248} C_VEL
LIN {X 0,Y 418.273,Z 388.389,A -85,B 0,C 180,E1 -10255.724,E2 -10255.724} C_VEL
LIN {X 0,Y 418.547,Z 394.535,A -85,B 0,C 180,E1 -10258.556,E2 -10258.556} C_VEL
LIN {X 0,Y 418.284,Z 400.924,A -85,B 0,C 180,E1 -10261.444,E2 -10261.444} C_VEL
LIN {X 0,Y 418.089,Z 409.026,A -85,B 0,C 180,E1 -10265.304,E2 -10265.304} C_VEL
LIN {X 0,Y 417.922,Z 415.221,A -85,B 0,C 180,E1 -10268.218,E2 -10268.218} C_VEL
LIN {X 0,Y 417.742,Z 423.385,A -85,B 0,C 180,E1 -10272.128,E2 -10272.128} C_VEL
LIN {X 0,Y 417.653,Z 426.501,A -85,B 0,C 180,E1 -10273.626,E2 -10273.626} C_VEL
LIN {X 0,Y 420.901,Z 440.701,A -85,B 0,C 180,E1 -10274.282,E2 -10274.282} C_VEL
LIN {X 0,Y 422.347,Z 449.401,A -85,B 0,C 180,E1 -10274.762,E2 -10274.762} C_VEL
LIN {X 0,Y 421.696,Z 461.374,A -85,B 0,C 180,E1 -10275.465,E2 -10275.465} C_VEL
LIN {X 0,Y 420.981,Z 473.086,A -85,B 0,C 180,E1 -10276.362,E2 -10276.362} C_VEL
LIN {X 0,Y 420.207,Z 483.958,A -85,B 0,C 180,E1 -10277.417,E2 -10277.417} C_VEL
LIN {X 0,Y 419.51,Z 493.514,A -85,B 0,C 180,E1 -10278.56,E2 -10278.56} C_VEL
LIN {X 0,Y 418.792,Z 503.084,A -85,B 0,C 180,E1 -10279.985,E2 -10279.985} C_VEL
LIN {X 0,Y 418.195,Z 510.948,A -85,B 0,C 180,E1 -10281.439,E2 -10281.439} C_VEL
LIN {X 0,Y 417.737,Z 517.767,A -85,B 0,C 180,E1 -10283.026,E2 -10283.026} C_VEL
LIN {X 0,Y 417.384,Z 522.986,A -85,B 0,C 180,E1 -10284.594,E2 -10284.594} C_VEL
LIN {X 0,Y 417.202,Z 526.502,A -85,B 0,C 180,E1 -10285.975,E2 -10285.975} C_VEL
LIN {X 0,Y 417.074,Z 528.63,A -85,B 0,C 180,E1 -10287.063,E2 -10287.063} C_VEL
LIN {X 0,Y 416.93,Z 530.867,A -85,B 0,C 180,E1 -10288.77,E2 -10288.77} C_VEL
LIN {X 0,Y 416.841,Z 531.838,A -85,B 0,C 180,E1 -10290.697,E2 -10290.697} C_VEL
LIN {X 0,Y 416.886,Z 531.288,A -85,B 0,C 180,E1 -10292.549,E2 -10292.549} C_VEL
LIN {X 0,Y 416.966,Z 529.331,A -85,B 0,C 180,E1 -10294.318,E2 -10294.318} C_VEL
LIN {X 0,Y 417.198,Z 525.894,A -85,B 0,C 180,E1 -10296.128,E2 -10296.128} C_VEL
LIN {X 0,Y 417.43,Z 521.617,A -85,B 0,C 180,E1 -10297.69,E2 -10297.69} C_VEL
LIN {X 0,Y 417.696,Z 515.841,A -85,B 0,C 180,E1 -10299.286,E2 -10299.286} C_VEL
LIN {X 0,Y 418.165,Z 508.584,A -85,B 0,C 180,E1 -10300.859,E2 -10300.859} C_VEL
LIN {X 0,Y 418.662,Z 500.99,A -85,B 0,C 180,E1 -10302.18,E2 -10302.18} C_VEL
LIN {X 0,Y 419.338,Z 491.3,A -85,B 0,C 180,E1 -10303.541,E2 -10303.541} C_VEL
LIN {X 0,Y 419.984,Z 481.568,A -85,B 0,C 180,E1 -10304.654,E2 -10304.654} C_VEL
LIN {X 0,Y 420.629,Z 471.232,A -85,B 0,C 180,E1 -10305.614,E2 -10305.614} C_VEL
LIN {X 0,Y 421.299,Z 458.758,A -85,B 0,C 180,E1 -10306.523,E2 -10306.523} C_VEL
LIN {X 0,Y 421.854,Z 448.605,A -85,B 0,C 180,E1 -10307.095,E2 -10307.095} C_VEL
LIN {X 0,Y 419.422,Z 435.265,A -85,B 0,C 180,E1 -10307.763,E2 -10307.763} C_VEL
LIN {X 0,Y 417.533,Z 425.904,A -85,B 0,C 180,E1 -10308.125,E2 -10308.125} C_VEL
LIN {X 0,Y 417.64,Z 419.012,A -85,B 0,C 180,E1 -10311.49,E2 -10311.49} C_VEL
LIN {X 0,Y 417.863,Z 411.577,A -85,B 0,C 180,E1 -10315.12,E2 -10315.12} C_VEL
LIN {X 0,Y 418.008,Z 404.497,A -85,B 0,C 180,E1 -10318.585,E2 -10318.585} C_VEL
LIN {X 0,Y 418.145,Z 398.673,A -85,B 0,C 180,E1 -10321.433,E2 -10321.433} C_VEL
LIN {X 0,Y 418.329,Z 391.069,A -85,B 0,C 180,E1 -10325.163,E2 -10325.163} C_VEL
LIN {X 0,Y 418.356,Z 388.375,A -85,B 0,C 180,E1 -10326.484,E2 -10326.484} C_VEL
LIN {X 0,Y 418.285,Z 388.385,A -85,B 0,C 180,E1 -10330.363,E2 -10330.363} C_VEL
LIN {X 0,Y 418.318,Z 388.379,A -85,B 0,C 180,E1 -10333.403,E2 -10333.403} C_VEL
LIN {X 0,Y 418.348,Z 388.376,A -85,B 0,C 180,E1 -10336.997,E2 -10336.997} C_VEL
LIN {X 0,Y 418.34,Z 388.375,A -85,B 0,C 180,E1 -10340.327,E2 -10340.327} C_VEL
LIN {X 0,Y 418.459,Z 388.364,A -85,B 0,C 180,E1 -10343.246,E2 -10343.246} C_VEL
LIN {X 0,Y 418.325,Z 388.38,A -85,B 0,C 180,E1 -10345.179,E2 -10345.179} C_VEL
LIN {X 0,Y 418.534,Z 388.353,A -85,B 0,C 180,E1 -10348.073,E2 -10348.073} C_VEL
LIN {X 0,Y 418.501,Z 388.378,A -85,B 0,C 180,E1 -10349.036,E2 -10349.036} C_VEL
LIN {X 0,Y 418.797,Z 389.897,A -85,B 0,C 180,E1 -10349.998,E2 -10349.998} C_VEL
LIN {X 0,Y 418.702,Z 391.004,A -85,B 0,C 180,E1 -10350.675,E2 -10350.675} C_VEL
LIN {X 0,Y 417.939,Z 392.383,A -85,B 0,C 180,E1 -10351.454,E2 -10351.454} C_VEL
LIN {X 0,Y 414.875,Z 394.865,A -85,B 0,C 180,E1 -10352.706,E2 -10352.706} C_VEL
LIN {X 0,Y 412.335,Z 396.873,A -85,B 0,C 180,E1 -10353.717,E2 -10353.717} C_VEL
LIN {X 0,Y 411.278,Z 398.312,A -85,B 0,C 180,E1 -10354.504,E2 -10354.504} C_VEL
LIN {X 0,Y 411.21,Z 398.765,A -85,B 0,C 180,E1 -10354.773,E2 -10354.773} C_VEL
LIN {X 0,Y 411.055,Z 403.953,A -85,B 0,C 180,E1 -10357.859,E2 -10357.859} C_VEL
LIN {X 0,Y 410.796,Z 409.039,A -85,B 0,C 180,E1 -10360.845,E2 -10360.845} C_VEL
LIN {X 0,Y 410.708,Z 412.498,A -85,B 0,C 180,E1 -10362.851,E2 -10362.851} C_VEL
LIN {X 0,Y 410.441,Z 418.848,A -85,B 0,C 180,E1 -10366.487,E2 -10366.487} C_VEL
LIN {X 0,Y 410.32,Z 423.105,A -85,B 0,C 180,E1 -10368.892,E2 -10368.892} C_VEL
LIN {X 0,Y 412.717,Z 435.618,A -85,B 0,C 180,E1 -10369.481,E2 -10369.481} C_VEL
LIN {X 0,Y 413.757,Z 442.989,A -85,B 0,C 180,E1 -10369.92,E2 -10369.92} C_VEL
LIN {X 0,Y 413.178,Z 454.973,A -85,B 0,C 180,E1 -10370.765,E2 -10370.765} C_VEL
LIN {X 0,Y 412.552,Z 465.383,A -85,B 0,C 180,E1 -10371.745,E2 -10371.745} C_VEL
LIN {X 0,Y 412.018,Z 474.185,A -85,B 0,C 180,E1 -10372.799,E2 -10372.799} C_VEL
LIN {X 0,Y 411.509,Z 481.736,A -85,B 0,C 180,E1 -10373.927,E2 -10373.927} C_VEL
LIN {X 0,Y 411.032,Z 489.066,A -85,B 0,C 180,E1 -10375.303,E2 -10375.303} C_VEL
LIN {X 0,Y 410.626,Z 495.068,A -85,B 0,C 180,E1 -10376.76,E2 -10376.76} C_VEL
LIN {X 0,Y 410.364,Z 499.25,A -85,B 0,C 180,E1 -10378.094,E2 -10378.094} C_VEL
LIN {X 0,Y 410.182,Z 502.997,A -85,B 0,C 180,E1 -10379.791,E2 -10379.791} C_VEL
LIN {X 0,Y 410.01,Z 504.721,A -85,B 0,C 180,E1 -10381.014,E2 -10381.014} C_VEL
LIN {X 0,Y 409.932,Z 505.596,A -85,B 0,C 180,E1 -10382.102,E2 -10382.102} C_VEL
LIN {X 0,Y 409.926,Z 505.88,A -85,B 0,C 180,E1 -10383.269,E2 -10383.269} C_VEL
LIN {X 0,Y 410.006,Z 505.324,A -85,B 0,C 180,E1 -10384.637,E2 -10384.637} C_VEL
LIN {X 0,Y 410.195,Z 503.273,A -85,B 0,C 180,E1 -10386.365,E2 -10386.365} C_VEL
LIN {X 0,Y 410.466,Z 499.691,A -85,B 0,C 180,E1 -10388.049,E2 -10388.049} C_VEL
LIN {X 0,Y 410.836,Z 494.647,A -85,B 0,C 180,E1 -10389.665,E2 -10389.665} C_VEL
LIN {X 0,Y 411.187,Z 489.669,A -85,B 0,C 180,E1 -10390.88,E2 -10390.88} C_VEL
LIN {X 0,Y 411.594,Z 483.573,A -85,B 0,C 180,E1 -10392.078,E2 -10392.078} C_VEL
LIN {X 0,Y 412.143,Z 475.486,A -85,B 0,C 180,E1 -10393.338,E2 -10393.338} C_VEL
LIN {X 0,Y 412.783,Z 467.377,A -85,B 0,C 180,E1 -10394.35,E2 -10394.35} C_VEL
LIN {X 0,Y 413.314,Z 459.081,A -85,B 0,C 180,E1 -10395.189,E2 -10395.189} C_VEL
LIN {X 0,Y 413.935,Z 448.246,A -85,B 0,C 180,E1 -10396.048,E2 -10396.048} C_VEL
LIN {X 0,Y 414.108,Z 442.585,A -85,B 0,C 180,E1 -10396.413,E2 -10396.413} C_VEL
LIN {X 0,Y 411.949,Z 430.515,A -85,B 0,C 180,E1 -10397.114,E2 -10397.114} C_VEL
LIN {X 0,Y 410.477,Z 423.655,A -85,B 0,C 180,E1 -10397.436,E2 -10397.436} C_VEL
LIN {X 0,Y 410.634,Z 416.943,A -85,B 0,C 180,E1 -10401.341,E2 -10401.341} C_VEL
LIN {X 0,Y 410.843,Z 411.679,A -85,B 0,C 180,E1 -10404.436,E2 -10404.436} C_VEL
LIN {X 0,Y 411.031,Z 405.77,A -85,B 0,C 180,E1 -10407.991,E2 -10407.991} C_VEL
LIN {X 0,Y 411.344,Z 400.123,A -85,B 0,C 180,E1 -10411.42,E2 -10411.42} C_VEL
LIN {X 0,Y 411.622,Z 394.701,A -85,B 0,C 180,E1 -10414.804,E2 -10414.804} C_VEL
LIN {X 0,Y 411.468,Z 390.893,A -85,B 0,C 180,E1 -10417.261,E2 -10417.261} C_VEL
LIN {X 0,Y 411.237,Z 389.263,A -85,B 0,C 180,E1 -10418.443,E2 -10418.443} C_VEL
LIN {X 0,Y 411.213,Z 389.269,A -85,B 0,C 180,E1 -10421.051,E2 -10421.051} C_VEL
LIN {X 0,Y 411.232,Z 389.265,A -85,B 0,C 180,E1 -10424.131,E2 -10424.131} C_VEL
LIN {X 0,Y 411.292,Z 389.255,A -85,B 0,C 180,E1 -10427.166,E2 -10427.166} C_VEL
LIN {X 0,Y 411.289,Z 389.255,A -85,B 0,C 180,E1 -10430.161,E2 -10430.161} C_VEL
LIN {X 0,Y 411.438,Z 389.237,A -85,B 0,C 180,E1 -10433.133,E2 -10433.133} C_VEL
LIN {X 0,Y 411.298,Z 389.255,A -85,B 0,C 180,E1 -10435.099,E2 -10435.099} C_VEL
LIN {X 0,Y 411.492,Z 389.228,A -85,B 0,C 180,E1 -10438.043,E2 -10438.043} C_VEL
LIN {X 0,Y 411.621,Z 389.213,A -85,B 0,C 180,E1 -10440,E2 -10440} C_VEL
LIN {X 0,Y 411.452,Z 389.234,A -85,B 0,C 180,E1 -10442.938,E2 -10442.938} C_VEL
LIN {X 0,Y 411.47,Z 389.231,A -85,B 0,C 180,E1 -10445.882,E2 -10445.882} C_VEL
LIN {X 0,Y 411.458,Z 389.233,A -85,B 0,C 180,E1 -10447.854,E2 -10447.854} C_VEL
LIN {X 0,Y 411.283,Z 389.253,A -85,B 0,C 180,E1 -10451.833,E2 -10451.833} C_VEL
LIN {X 0,Y 411.247,Z 389.259,A -85,B 0,C 180,E1 -10454.853,E2 -10454.853} C_VEL
LIN {X 0,Y 411.234,Z 389.26,A -85,B 0,C 180,E1 -10457.916,E2 -10457.916} C_VEL
LIN {X 0,Y 411.217,Z 389.26,A -85,B 0,C 180,E1 -10461.033,E2 -10461.033} C_VEL
LIN {X 0,Y 411.208,Z 389.261,A -85,B 0,C 180,E1 -10464.217,E2 -10464.217} C_VEL
LIN {X 0,Y 411.24,Z 389.258,A -85,B 0,C 180,E1 -10467.479,E2 -10467.479} C_VEL
LIN {X 0,Y 411.179,Z 389.267,A -85,B 0,C 180,E1 -10470.849,E2 -10470.849} C_VEL
LIN {X 0,Y 411.188,Z 389.267,A -85,B 0,C 180,E1 -10474.336,E2 -10474.336} C_VEL
LIN {X 0,Y 411.188,Z 389.268,A -85,B 0,C 180,E1 -10477.975,E2 -10477.975} C_VEL
LIN {X 0,Y 411.195,Z 389.266,A -85,B 0,C 180,E1 -10481.238,E2 -10481.238} C_VEL
LIN {X 0,Y 411.222,Z 389.264,A -85,B 0,C 180,E1 -10484.484,E2 -10484.484} C_VEL
LIN {X 0,Y 411.22,Z 389.262,A -85,B 0,C 180,E1 -10487.299,E2 -10487.299} C_VEL
LIN {X 0,Y 411.22,Z 389.264,A -85,B 0,C 180,E1 -10490.78,E2 -10490.78} C_VEL
LIN {X 0,Y 411.194,Z 389.297,A -85,B 0,C 180,E1 -10492.03,E2 -10492.03} C_VEL
LIN {X 0,Y 412.734,Z 396.767,A -85,B 0,C 180,E1 -10495.355,E2 -10495.355} C_VEL
LIN {X 0,Y 413.983,Z 403.792,A -85,B 0,C 180,E1 -10498.249,E2 -10498.249} C_VEL
LIN {X 0,Y 414.013,Z 408.385,A -85,B 0,C 180,E1 -10499.968,E2 -10499.968} C_VEL
LIN {X 0,Y 412.878,Z 418.988,A -85,B 0,C 180,E1 -10503.735,E2 -10503.735} C_VEL
LIN {X 0,Y 412.045,Z 428.824,A -85,B 0,C 180,E1 -10507.08,E2 -10507.08} C_VEL
LIN {X 0,Y 411.332,Z 439.329,A -85,B 0,C 180,E1 -10510.541,E2 -10510.541} C_VEL
LIN {X 0,Y 410.981,Z 446.225,A -85,B 0,C 180,E1 -10512.766,E2 -10512.766} C_VEL
LIN {X 0,Y 413.047,Z 459.766,A -85,B 0,C 180,E1 -10513.24,E2 -10513.24} C_VEL
LIN {X 0,Y 414.294,Z 472.392,A -85,B 0,C 180,E1 -10513.86,E2 -10513.86} C_VEL
LIN {X 0,Y 413.854,Z 482.914,A -85,B 0,C 180,E1 -10514.489,E2 -10514.489} C_VEL
LIN {X 0,Y 413.09,Z 494.111,A -85,B 0,C 180,E1 -10515.343,E2 -10515.343} C_VEL
LIN {X 0,Y 412.368,Z 504.858,A -85,B 0,C 180,E1 -10516.381,E2 -10516.381} C_VEL
LIN {X 0,Y 411.745,Z 515.608,A -85,B 0,C 180,E1 -10517.683,E2 -10517.683} C_VEL
LIN {X 0,Y 411.135,Z 524.025,A -85,B 0,C 180,E1 -10518.915,E2 -10518.915} C_VEL
LIN {X 0,Y 410.654,Z 532.235,A -85,B 0,C 180,E1 -10520.397,E2 -10520.397} C_VEL
LIN {X 0,Y 410.361,Z 537.807,A -85,B 0,C 180,E1 -10521.632,E2 -10521.632} C_VEL
LIN {X 0,Y 410.094,Z 543.226,A -85,B 0,C 180,E1 -10523.112,E2 -10523.112} C_VEL
LIN {X 0,Y 410.026,Z 547.431,A -85,B 0,C 180,E1 -10524.593,E2 -10524.593} C_VEL
LIN {X 0,Y 409.959,Z 550.535,A -85,B 0,C 180,E1 -10526.07,E2 -10526.07} C_VEL
LIN {X 0,Y 409.959,Z 552.061,A -85,B 0,C 180,E1 -10527.054,E2 -10527.054} C_VEL
LIN {X 0,Y 410.041,Z 553.118,A -85,B 0,C 180,E1 -10528.038,E2 -10528.038} C_VEL
LIN {X 0,Y 409.982,Z 553.765,A -85,B 0,C 180,E1 -10529.02,E2 -10529.02} C_VEL
LIN {X 0,Y 409.949,Z 554.015,A -85,B 0,C 180,E1 -10530.002,E2 -10530.002} C_VEL
LIN {X 0,Y 409.984,Z 553.837,A -85,B 0,C 180,E1 -10530.984,E2 -10530.984} C_VEL
LIN {X 0,Y 410.05,Z 553.226,A -85,B 0,C 180,E1 -10531.967,E2 -10531.967} C_VEL
LIN {X 0,Y 409.958,Z 552.213,A -85,B 0,C 180,E1 -10532.95,E2 -10532.95} C_VEL
LIN {X 0,Y 409.961,Z 550.793,A -85,B 0,C 180,E1 -10533.934,E2 -10533.934} C_VEL
LIN {X 0,Y 410.036,Z 547.802,A -85,B 0,C 180,E1 -10535.411,E2 -10535.411} C_VEL
LIN {X 0,Y 410.167,Z 543.745,A -85,B 0,C 180,E1 -10536.891,E2 -10536.891} C_VEL
LIN {X 0,Y 410.448,Z 537.473,A -85,B 0,C 180,E1 -10538.619,E2 -10538.619} C_VEL
LIN {X 0,Y 410.831,Z 530.634,A -85,B 0,C 180,E1 -10540.101,E2 -10540.101} C_VEL
LIN {X 0,Y 411.296,Z 523.668,A -85,B 0,C 180,E1 -10541.335,E2 -10541.335} C_VEL
LIN {X 0,Y 411.945,Z 515.284,A -85,B 0,C 180,E1 -10542.565,E2 -10542.565} C_VEL
LIN {X 0,Y 412.594,Z 504.95,A -85,B 0,C 180,E1 -10543.798,E2 -10543.798} C_VEL
LIN {X 0,Y 413.431,Z 493.393,A -85,B 0,C 180,E1 -10544.901,E2 -10544.901} C_VEL
LIN {X 0,Y 414.26,Z 481.965,A -85,B 0,C 180,E1 -10545.752,E2 -10545.752} C_VEL
LIN {X 0,Y 414.536,Z 471.993,A -85,B 0,C 180,E1 -10546.352,E2 -10546.352} C_VEL
LIN {X 0,Y 413.227,Z 458.265,A -85,B 0,C 180,E1 -10547.035,E2 -10547.035} C_VEL
LIN {X 0,Y 410.991,Z 445.175,A -85,B 0,C 180,E1 -10547.553,E2 -10547.553} C_VEL
LIN {X 0,Y 411.613,Z 434.426,A -85,B 0,C 180,E1 -10551.014,E2 -10551.014} C_VEL
LIN {X 0,Y 412.45,Z 423.341,A -85,B 0,C 180,E1 -10554.677,E2 -10554.677} C_VEL
LIN {X 0,Y 413.419,Z 412.279,A -85,B 0,C 180,E1 -10558.426,E2 -10558.426} C_VEL
LIN {X 0,Y 414.032,Z 406.012,A -85,B 0,C 180,E1 -10560.615,E2 -10560.615} C_VEL
LIN {X 0,Y 413.542,Z 401.299,A -85,B 0,C 180,E1 -10562.367,E2 -10562.367} C_VEL
LIN {X 0,Y 412.027,Z 393.461,A -85,B 0,C 180,E1 -10565.448,E2 -10565.448} C_VEL
LIN {X 0,Y 411.216,Z 389.264,A -85,B 0,C 180,E1 -10567.201,E2 -10567.201} C_VEL
LIN {X 0,Y 411.165,Z 389.269,A -85,B 0,C 180,E1 -10570.508,E2 -10570.508} C_VEL
LIN {X 0,Y 411.169,Z 389.268,A -85,B 0,C 180,E1 -10574.119,E2 -10574.119} C_VEL
LIN {X 0,Y 411.174,Z 389.269,A -85,B 0,C 180,E1 -10577.307,E2 -10577.307} C_VEL
LIN {X 0,Y 411.186,Z 389.267,A -85,B 0,C 180,E1 -10580.772,E2 -10580.772} C_VEL
LIN {X 0,Y 411.201,Z 389.265,A -85,B 0,C 180,E1 -10584.471,E2 -10584.471} C_VEL
LIN {X 0,Y 411.212,Z 389.261,A -85,B 0,C 180,E1 -10586.874,E2 -10586.874} C_VEL
LIN {X 0,Y 411.216,Z 389.261,A -85,B 0,C 180,E1 -10590.65,E2 -10590.65} C_VEL
LIN {X 0,Y 411.17,Z 389.27,A -85,B 0,C 180,E1 -10593.614,E2 -10593.614} C_VEL
LIN {X 0,Y 411.193,Z 389.268,A -85,B 0,C 180,E1 -10596.851,E2 -10596.851} C_VEL
LIN {X 0,Y 411.221,Z 389.263,A -85,B 0,C 180,E1 -10600.051,E2 -10600.051} C_VEL
LIN {X 0,Y 411.27,Z 389.256,A -85,B 0,C 180,E1 -10603.131,E2 -10603.131} C_VEL
LIN {X 0,Y 411.312,Z 389.252,A -85,B 0,C 180,E1 -10606.896,E2 -10606.896} C_VEL
LIN {X 0,Y 411.285,Z 389.254,A -85,B 0,C 180,E1 -10610.161,E2 -10610.161} C_VEL
LIN {X 0,Y 411.396,Z 389.243,A -85,B 0,C 180,E1 -10613.132,E2 -10613.132} C_VEL
LIN {X 0,Y 411.267,Z 389.357,A -85,B 0,C 180,E1 -10615.528,E2 -10615.528} C_VEL
LIN {X 0,Y 411.568,Z 394.725,A -85,B 0,C 180,E1 -10618.043,E2 -10618.043} C_VEL
LIN {X 0,Y 411.408,Z 399.964,A -85,B 0,C 180,E1 -10620.489,E2 -10620.489} C_VEL
LIN {X 0,Y 411.098,Z 408.324,A -85,B 0,C 180,E1 -10624.412,E2 -10624.412} C_VEL
LIN {X 0,Y 410.984,Z 414.379,A -85,B 0,C 180,E1 -10627.325,E2 -10627.325} C_VEL
LIN {X 0,Y 410.743,Z 421.689,A -85,B 0,C 180,E1 -10630.848,E2 -10630.848} C_VEL
LIN {X 0,Y 410.635,Z 426.702,A -85,B 0,C 180,E1 -10633.28,E2 -10633.28} C_VEL
LIN {X 0,Y 414.058,Z 441.286,A -85,B 0,C 180,E1 -10633.978,E2 -10633.978} C_VEL
LIN {X 0,Y 415.525,Z 451.23,A -85,B 0,C 180,E1 -10634.547,E2 -10634.547} C_VEL
LIN {X 0,Y 414.882,Z 462.363,A -85,B 0,C 180,E1 -10635.229,E2 -10635.229} C_VEL
LIN {X 0,Y 414.123,Z 473.806,A -85,B 0,C 180,E1 -10636.134,E2 -10636.134} C_VEL
LIN {X 0,Y 413.278,Z 485.086,A -85,B 0,C 180,E1 -10637.26,E2 -10637.26} C_VEL
LIN {X 0,Y 412.59,Z 494.076,A -85,B 0,C 180,E1 -10638.368,E2 -10638.368} C_VEL
LIN {X 0,Y 411.902,Z 502.84,A -85,B 0,C 180,E1 -10639.693,E2 -10639.693} C_VEL
LIN {X 0,Y 411.195,Z 511.389,A -85,B 0,C 180,E1 -10641.296,E2 -10641.296} C_VEL
LIN {X 0,Y 410.733,Z 517.728,A -85,B 0,C 180,E1 -10642.797,E2 -10642.797} C_VEL
LIN {X 0,Y 410.372,Z 522.643,A -85,B 0,C 180,E1 -10644.269,E2 -10644.269} C_VEL
LIN {X 0,Y 410.148,Z 526.788,A -85,B 0,C 180,E1 -10645.909,E2 -10645.909} C_VEL
LIN {X 0,Y 409.948,Z 529.732,A -85,B 0,C 180,E1 -10647.573,E2 -10647.573} C_VEL
LIN {X 0,Y 409.816,Z 531.292,A -85,B 0,C 180,E1 -10649,E2 -10649} C_VEL
LIN {X 0,Y 409.745,Z 532.061,A -85,B 0,C 180,E1 -10650.968,E2 -10650.968} C_VEL
LIN {X 0,Y 409.791,Z 531.255,A -85,B 0,C 180,E1 -10652.82,E2 -10652.82} C_VEL
LIN {X 0,Y 409.884,Z 529.131,A -85,B 0,C 180,E1 -10654.61,E2 -10654.61} C_VEL
LIN {X 0,Y 410.124,Z 525.703,A -85,B 0,C 180,E1 -10656.349,E2 -10656.349} C_VEL
LIN {X 0,Y 410.377,Z 520.871,A -85,B 0,C 180,E1 -10658.062,E2 -10658.062} C_VEL
LIN {X 0,Y 410.737,Z 515.013,A -85,B 0,C 180,E1 -10659.646,E2 -10659.646} C_VEL
LIN {X 0,Y 411.229,Z 507.505,A -85,B 0,C 180,E1 -10661.237,E2 -10661.237} C_VEL
LIN {X 0,Y 411.839,Z 498.23,A -85,B 0,C 180,E1 -10662.793,E2 -10662.793} C_VEL
LIN {X 0,Y 412.601,Z 488.229,A -85,B 0,C 180,E1 -10664.126,E2 -10664.126} C_VEL
LIN {X 0,Y 413.269,Z 478.307,A -85,B 0,C 180,E1 -10665.199,E2 -10665.199} C_VEL
LIN {X 0,Y 413.927,Z 467.905,A -85,B 0,C 180,E1 -10666.114,E2 -10666.114} C_VEL
LIN {X 0,Y 414.576,Z 456.618,A -85,B 0,C 180,E1 -10666.902,E2 -10666.902} C_VEL
LIN {X 0,Y 414.854,Z 448.821,A -85,B 0,C 180,E1 -10667.339,E2 -10667.339} C_VEL
LIN {X 0,Y 412.376,Z 435.405,A -85,B 0,C 180,E1 -10668.027,E2 -10668.027} C_VEL
LIN {X 0,Y 410.475,Z 426.039,A -85,B 0,C 180,E1 -10668.399,E2 -10668.399} C_VEL
LIN {X 0,Y 410.627,Z 418.804,A -85,B 0,C 180,E1 -10671.963,E2 -10671.963} C_VEL
LIN {X 0,Y 410.83,Z 411.352,A -85,B 0,C 180,E1 -10675.629,E2 -10675.629} C_VEL
LIN {X 0,Y 410.979,Z 404.255,A -85,B 0,C 180,E1 -10679.133,E2 -10679.133} C_VEL
LIN {X 0,Y 411.166,Z 397.419,A -85,B 0,C 180,E1 -10682.514,E2 -10682.514} C_VEL
LIN {X 0,Y 411.375,Z 390.754,A -85,B 0,C 180,E1 -10685.792,E2 -10685.792} C_VEL
LIN {X 0,Y 411.325,Z 389.251,A -85,B 0,C 180,E1 -10686.592,E2 -10686.592} C_VEL
LIN {X 0,Y 411.217,Z 389.263,A -85,B 0,C 180,E1 -10690.049,E2 -10690.049} C_VEL
LIN {X 0,Y 411.265,Z 389.256,A -85,B 0,C 180,E1 -10693.129,E2 -10693.129} C_VEL
LIN {X 0,Y 411.307,Z 389.254,A -85,B 0,C 180,E1 -10696.894,E2 -10696.894} C_VEL
LIN {X 0,Y 411.292,Z 389.254,A -85,B 0,C 180,E1 -10700.159,E2 -10700.159} C_VEL
LIN {X 0,Y 411.424,Z 389.24,A -85,B 0,C 180,E1 -10703.13,E2 -10703.13} C_VEL
LIN {X 0,Y 411.296,Z 389.256,A -85,B 0,C 180,E1 -10705.097,E2 -10705.097} C_VEL
LIN {X 0,Y 411.503,Z 389.229,A -85,B 0,C 180,E1 -10708.04,E2 -10708.04} C_VEL
LIN {X 0,Y 411.495,Z 389.422,A -85,B 0,C 180,E1 -10709.019,E2 -10709.019} C_VEL
LIN {X 0,Y 411.77,Z 390.949,A -85,B 0,C 180,E1 -10709.998,E2 -10709.998} C_VEL
LIN {X 0,Y 411.384,Z 395.728,A -85,B 0,C 180,E1 -10712.936,E2 -10712.936} C_VEL
LIN {X 0,Y 411.21,Z 398.765,A -85,B 0,C 180,E1 -10714.773,E2 -10714.773} C_VEL
LIN {X 0,Y 410.565,Z 400.175,A -85,B 0,C 180,E1 -10715.567,E2 -10715.567} C_VEL
LIN {X 0,Y 407.621,Z 402.703,A -85,B 0,C 180,E1 -10716.846,E2 -10716.846} C_VEL
LIN {X 0,Y 405.092,Z 404.741,A -85,B 0,C 180,E1 -10717.879,E2 -10717.879} C_VEL
LIN {X 0,Y 403.995,Z 406.214,A -85,B 0,C 180,E1 -10718.682,E2 -10718.682} C_VEL
LIN {X 0,Y 403.902,Z 406.683,A -85,B 0,C 180,E1 -10718.956,E2 -10718.956} C_VEL
LIN {X 0,Y 403.658,Z 413.254,A -85,B 0,C 180,E1 -10722.839,E2 -10722.839} C_VEL
LIN {X 0,Y 403.363,Z 419.777,A -85,B 0,C 180,E1 -10726.607,E2 -10726.607} C_VEL
LIN {X 0,Y 403.242,Z 423.327,A -85,B 0,C 180,E1 -10728.642,E2 -10728.642} C_VEL
LIN {X 0,Y 405.462,Z 434.512,A -85,B 0,C 180,E1 -10729.16,E2 -10729.16} C_VEL
LIN {X 0,Y 406.818,Z 444.184,A -85,B 0,C 180,E1 -10729.749,E2 -10729.749} C_VEL
LIN {X 0,Y 406.313,Z 454.761,A -85,B 0,C 180,E1 -10730.511,E2 -10730.511} C_VEL
LIN {X 0,Y 405.653,Z 464.919,A -85,B 0,C 180,E1 -10731.466,E2 -10731.466} C_VEL
LIN {X 0,Y 405.131,Z 473.104,A -85,B 0,C 180,E1 -10732.433,E2 -10732.433} C_VEL
LIN {X 0,Y 404.615,Z 480.726,A -85,B 0,C 180,E1 -10733.544,E2 -10733.544} C_VEL
LIN {X 0,Y 404.072,Z 488.382,A -85,B 0,C 180,E1 -10734.948,E2 -10734.948} C_VEL
LIN {X 0,Y 403.662,Z 494.336,A -85,B 0,C 180,E1 -10736.354,E2 -10736.354} C_VEL
LIN {X 0,Y 403.392,Z 498.599,A -85,B 0,C 180,E1 -10737.649,E2 -10737.649} C_VEL
LIN {X 0,Y 403.194,Z 502.41,A -85,B 0,C 180,E1 -10739.21,E2 -10739.21} C_VEL
LIN {X 0,Y 403.005,Z 504.371,A -85,B 0,C 180,E1 -10740.376,E2 -10740.376} C_VEL
LIN {X 0,Y 402.877,Z 505.641,A -85,B 0,C 180,E1 -10741.553,E2 -10741.553} C_VEL
LIN {X 0,Y 402.845,Z 506.304,A -85,B 0,C 180,E1 -10743.134,E2 -10743.134} C_VEL
LIN {X 0,Y 402.969,Z 505.528,A -85,B 0,C 180,E1 -10744.945,E2 -10744.945} C_VEL
LIN {X 0,Y 403.177,Z 503.24,A -85,B 0,C 180,E1 -10746.693,E2 -10746.693} C_VEL
LIN {X 0,Y 403.376,Z 500.524,A -85,B 0,C 180,E1 -10747.986,E2 -10747.986} C_VEL
LIN {X 0,Y 403.744,Z 496.379,A -85,B 0,C 180,E1 -10749.424,E2 -10749.424} C_VEL
LIN {X 0,Y 404.088,Z 491.557,A -85,B 0,C 180,E1 -10750.704,E2 -10750.704} C_VEL
LIN {X 0,Y 404.543,Z 484.902,A -85,B 0,C 180,E1 -10752.088,E2 -10752.088} C_VEL
LIN {X 0,Y 405.049,Z 478.124,A -85,B 0,C 180,E1 -10753.219,E2 -10753.219} C_VEL
LIN {X 0,Y 405.732,Z 469.53,A -85,B 0,C 180,E1 -10754.367,E2 -10754.367} C_VEL
LIN {X 0,Y 406.366,Z 460.498,A -85,B 0,C 180,E1 -10755.332,E2 -10755.332} C_VEL
LIN {X 0,Y 407.029,Z 449.739,A -85,B 0,C 180,E1 -10756.224,E2 -10756.224} C_VEL
LIN {X 0,Y 407.308,Z 444.382,A -85,B 0,C 180,E1 -10756.585,E2 -10756.585} C_VEL
LIN {X 0,Y 405.496,Z 433.49,A -85,B 0,C 180,E1 -10757.26,E2 -10757.26} C_VEL
LIN {X 0,Y 403.43,Z 423.889,A -85,B 0,C 180,E1 -10757.754,E2 -10757.754} C_VEL
LIN {X 0,Y 403.59,Z 417.396,A -85,B 0,C 180,E1 -10761.588,E2 -10761.588} C_VEL
LIN {X 0,Y 403.835,Z 411.76,A -85,B 0,C 180,E1 -10764.949,E2 -10764.949} C_VEL
LIN {X 0,Y 404.062,Z 405.907,A -85,B 0,C 180,E1 -10768.547,E2 -10768.547} C_VEL
LIN {X 0,Y 404.377,Z 400.332,A -85,B 0,C 180,E1 -10772.014,E2 -10772.014} C_VEL
LIN {X 0,Y 404.622,Z 395.018,A -85,B 0,C 180,E1 -10775.364,E2 -10775.364} C_VEL
LIN {X 0,Y 404.429,Z 391.756,A -85,B 0,C 180,E1 -10777.524,E2 -10777.524} C_VEL
LIN {X 0,Y 404.187,Z 390.141,A -85,B 0,C 180,E1 -10778.717,E2 -10778.717} C_VEL
LIN {X 0,Y 404.19,Z 390.144,A -85,B 0,C 180,E1 -10781.761,E2 -10781.761} C_VEL
LIN {X 0,Y 404.185,Z 390.142,A -85,B 0,C 180,E1 -10784.882,E2 -10784.882} C_VEL
LIN {X 0,Y 404.251,Z 390.131,A -85,B 0,C 180,E1 -10787.959,E2 -10787.959} C_VEL
LIN {X 0,Y 404.409,Z 390.11,A -85,B 0,C 180,E1 -10792.099,E2 -10792.099} C_VEL
LIN {X 0,Y 404.415,Z 390.111,A -85,B 0,C 180,E1 -10794.015,E2 -10794.015} C_VEL
LIN {X 0,Y 404.461,Z 390.104,A -85,B 0,C 180,E1 -10798.009,E2 -10798.009} C_VEL
LIN {X 0,Y 404.591,Z 390.088,A -85,B 0,C 180,E1 -10800,E2 -10800} C_VEL
LIN {X 0,Y 404.409,Z 390.112,A -85,B 0,C 180,E1 -10802.989,E2 -10802.989} C_VEL
LIN {X 0,Y 404.416,Z 390.109,A -85,B 0,C 180,E1 -10805.985,E2 -10805.985} C_VEL
LIN {X 0,Y 404.399,Z 390.112,A -85,B 0,C 180,E1 -10807.992,E2 -10807.992} C_VEL
LIN {X 0,Y 404.252,Z 390.129,A -85,B 0,C 180,E1 -10812.042,E2 -10812.042} C_VEL
LIN {X 0,Y 404.192,Z 390.136,A -85,B 0,C 180,E1 -10815.119,E2 -10815.119} C_VEL
LIN {X 0,Y 404.194,Z 390.134,A -85,B 0,C 180,E1 -10818.239,E2 -10818.239} C_VEL
LIN {X 0,Y 404.173,Z 390.136,A -85,B 0,C 180,E1 -10821.418,E2 -10821.418} C_VEL
LIN {X 0,Y 404.195,Z 390.137,A -85,B 0,C 180,E1 -10825.298,E2 -10825.298} C_VEL
LIN {X 0,Y 404.178,Z 390.139,A -85,B 0,C 180,E1 -10828.001,E2 -10828.001} C_VEL
LIN {X 0,Y 404.124,Z 390.145,A -85,B 0,C 180,E1 -10831.561,E2 -10831.561} C_VEL
LIN {X 0,Y 404.168,Z 390.141,A -85,B 0,C 180,E1 -10835.018,E2 -10835.018} C_VEL
LIN {X 0,Y 404.148,Z 390.143,A -85,B 0,C 180,E1 -10838.758,E2 -10838.758} C_VEL
LIN {X 0,Y 404.176,Z 390.141,A -85,B 0,C 180,E1 -10841.613,E2 -10841.613} C_VEL
LIN {X 0,Y 404.187,Z 390.141,A -85,B 0,C 180,E1 -10844.533,E2 -10844.533} C_VEL
LIN {X 0,Y 404.198,Z 390.137,A -85,B 0,C 180,E1 -10847.308,E2 -10847.308} C_VEL
LIN {X 0,Y 404.157,Z 390.143,A -85,B 0,C 180,E1 -10849.958,E2 -10849.958} C_VEL
LIN {X 0,Y 404.17,Z 390.177,A -85,B 0,C 180,E1 -10851.577,E2 -10851.577} C_VEL
LIN {X 0,Y 405.742,Z 397.967,A -85,B 0,C 180,E1 -10855.141,E2 -10855.141} C_VEL
LIN {X 0,Y 406.881,Z 404.294,A -85,B 0,C 180,E1 -10857.82,E2 -10857.82} C_VEL
LIN {X 0,Y 407.197,Z 408.063,A -85,B 0,C 180,E1 -10859.314,E2 -10859.314} C_VEL
LIN {X 0,Y 406.136,Z 417.431,A -85,B 0,C 180,E1 -10862.708,E2 -10862.708} C_VEL
LIN {X 0,Y 405.293,Z 426.596,A -85,B 0,C 180,E1 -10865.955,E2 -10865.955} C_VEL
LIN {X 0,Y 404.437,Z 437.562,A -85,B 0,C 180,E1 -10869.666,E2 -10869.666} C_VEL
LIN {X 0,Y 403.929,Z 445.965,A -85,B 0,C 180,E1 -10872.446,E2 -10872.446} C_VEL
LIN {X 0,Y 406.198,Z 460.51,A -85,B 0,C 180,E1 -10872.994,E2 -10872.994} C_VEL
LIN {X 0,Y 407.433,Z 473.61,A -85,B 0,C 180,E1 -10873.673,E2 -10873.673} C_VEL
LIN {X 0,Y 406.888,Z 484.303,A -85,B 0,C 180,E1 -10874.345,E2 -10874.345} C_VEL
LIN {X 0,Y 406.102,Z 495.17,A -85,B 0,C 180,E1 -10875.213,E2 -10875.213} C_VEL
LIN {X 0,Y 405.359,Z 505.303,A -85,B 0,C 180,E1 -10876.234,E2 -10876.234} C_VEL
LIN {X 0,Y 404.756,Z 515.167,A -85,B 0,C 180,E1 -10877.467,E2 -10877.467} C_VEL
LIN {X 0,Y 404.003,Z 525.107,A -85,B 0,C 180,E1 -10878.971,E2 -10878.971} C_VEL
LIN {X 0,Y 403.556,Z 533.103,A -85,B 0,C 180,E1 -10880.479,E2 -10880.479} C_VEL
LIN {X 0,Y 403.203,Z 539.449,A -85,B 0,C 180,E1 -10881.987,E2 -10881.987} C_VEL
LIN {X 0,Y 402.961,Z 544.61,A -85,B 0,C 180,E1 -10883.543,E2 -10883.543} C_VEL
LIN {X 0,Y 402.942,Z 548.318,A -85,B 0,C 180,E1 -10884.999,E2 -10884.999} C_VEL
LIN {X 0,Y 402.877,Z 550.286,A -85,B 0,C 180,E1 -10886.001,E2 -10886.001} C_VEL
LIN {X 0,Y 402.858,Z 551.827,A -85,B 0,C 180,E1 -10887.002,E2 -10887.002} C_VEL
LIN {X 0,Y 402.948,Z 552.901,A -85,B 0,C 180,E1 -10888.003,E2 -10888.003} C_VEL
LIN {X 0,Y 402.907,Z 553.558,A -85,B 0,C 180,E1 -10889.003,E2 -10889.003} C_VEL
LIN {X 0,Y 402.873,Z 553.817,A -85,B 0,C 180,E1 -10890.002,E2 -10890.002} C_VEL
LIN {X 0,Y 402.909,Z 553.659,A -85,B 0,C 180,E1 -10891.002,E2 -10891.002} C_VEL
LIN {X 0,Y 402.956,Z 553.056,A -85,B 0,C 180,E1 -10892.001,E2 -10892.001} C_VEL
LIN {X 0,Y 402.879,Z 550.641,A -85,B 0,C 180,E1 -10894.003,E2 -10894.003} C_VEL
LIN {X 0,Y 402.936,Z 547.664,A -85,B 0,C 180,E1 -10895.507,E2 -10895.507} C_VEL
LIN {X 0,Y 403.079,Z 543.625,A -85,B 0,C 180,E1 -10897.013,E2 -10897.013} C_VEL
LIN {X 0,Y 403.389,Z 537.374,A -85,B 0,C 180,E1 -10898.771,E2 -10898.771} C_VEL
LIN {X 0,Y 403.82,Z 530.555,A -85,B 0,C 180,E1 -10900.278,E2 -10900.278} C_VEL
LIN {X 0,Y 404.46,Z 522.101,A -85,B 0,C 180,E1 -10901.783,E2 -10901.783} C_VEL
LIN {X 0,Y 405.233,Z 511.845,A -85,B 0,C 180,E1 -10903.237,E2 -10903.237} C_VEL
LIN {X 0,Y 405.923,Z 501.932,A -85,B 0,C 180,E1 -10904.375,E2 -10904.375} C_VEL
LIN {X 0,Y 406.824,Z 490.623,A -85,B 0,C 180,E1 -10905.405,E2 -10905.405} C_VEL
LIN {X 0,Y 407.645,Z 478.8,A -85,B 0,C 180,E1 -10906.252,E2 -10906.252} C_VEL
LIN {X 0,Y 407.764,Z 472.983,A -85,B 0,C 180,E1 -10906.605,E2 -10906.605} C_VEL
LIN {X 0,Y 406.573,Z 459.817,A -85,B 0,C 180,E1 -10907.296,E2 -10907.296} C_VEL
LIN {X 0,Y 404.316,Z 446.88,A -85,B 0,C 180,E1 -10907.829,E2 -10907.829} C_VEL
LIN {X 0,Y 403.975,Z 444.668,A -85,B 0,C 180,E1 -10907.926,E2 -10907.926} C_VEL
LIN {X 0,Y 404.635,Z 434.164,A -85,B 0,C 180,E1 -10911.394,E2 -10911.394} C_VEL
LIN {X 0,Y 405.508,Z 423.082,A -85,B 0,C 180,E1 -10915.128,E2 -10915.128} C_VEL
LIN {X 0,Y 406.581,Z 412.078,A -85,B 0,C 180,E1 -10918.948,E2 -10918.948} C_VEL
LIN {X 0,Y 407.07,Z 407.216,A -85,B 0,C 180,E1 -10920.681,E2 -10920.681} C_VEL
LIN {X 0,Y 406.604,Z 402.673,A -85,B 0,C 180,E1 -10922.402,E2 -10922.402} C_VEL
LIN {X 0,Y 405.158,Z 395.23,A -85,B 0,C 180,E1 -10925.385,E2 -10925.385} C_VEL
LIN {X 0,Y 404.155,Z 390.145,A -85,B 0,C 180,E1 -10927.571,E2 -10927.571} C_VEL
LIN {X 0,Y 404.124,Z 390.148,A -85,B 0,C 180,E1 -10930.076,E2 -10930.076} C_VEL
LIN {X 0,Y 404.147,Z 390.144,A -85,B 0,C 180,E1 -10933.082,E2 -10933.082} C_VEL
LIN {X 0,Y 404.127,Z 390.14,A -85,B 0,C 180,E1 -10935.923,E2 -10935.923} C_VEL
LIN {X 0,Y 404.109,Z 390.145,A -85,B 0,C 180,E1 -10938.633,E2 -10938.633} C_VEL
LIN {X 0,Y 404.147,Z 390.138,A -85,B 0,C 180,E1 -10941.495,E2 -10941.495} C_VEL
LIN {X 0,Y 404.185,Z 390.137,A -85,B 0,C 180,E1 -10944.984,E2 -10944.984} C_VEL
LIN {X 0,Y 404.145,Z 390.142,A -85,B 0,C 180,E1 -10948.443,E2 -10948.443} C_VEL
LIN {X 0,Y 404.155,Z 390.141,A -85,B 0,C 180,E1 -10950.862,E2 -10950.862} C_VEL
LIN {X 0,Y 404.157,Z 390.142,A -85,B 0,C 180,E1 -10954.723,E2 -10954.723} C_VEL
LIN {X 0,Y 404.172,Z 390.139,A -85,B 0,C 180,E1 -10957.508,E2 -10957.508} C_VEL
LIN {X 0,Y 404.172,Z 390.142,A -85,B 0,C 180,E1 -10960.708,E2 -10960.708} C_VEL
LIN {X 0,Y 404.228,Z 390.136,A -85,B 0,C 180,E1 -10963.848,E2 -10963.848} C_VEL
LIN {X 0,Y 404.29,Z 390.127,A -85,B 0,C 180,E1 -10966.939,E2 -10966.939} C_VEL
LIN {X 0,Y 404.253,Z 390.131,A -85,B 0,C 180,E1 -10969.988,E2 -10969.988} C_VEL
LIN {X 0,Y 404.346,Z 390.121,A -85,B 0,C 180,E1 -10973.011,E2 -10973.011} C_VEL
LIN {X 0,Y 404.25,Z 390.229,A -85,B 0,C 180,E1 -10975.263,E2 -10975.263} C_VEL
LIN {X 0,Y 404.505,Z 394.942,A -85,B 0,C 180,E1 -10977.51,E2 -10977.51} C_VEL
LIN {X 0,Y 404.47,Z 400.123,A -85,B 0,C 180,E1 -10980,E2 -10980} C_VEL
LIN {X 0,Y 404.084,Z 409.67,A -85,B 0,C 180,E1 -10984.489,E2 -10984.489} C_VEL
LIN {X 0,Y 403.965,Z 415.595,A -85,B 0,C 180,E1 -10987.399,E2 -10987.399} C_VEL
LIN {X 0,Y 403.698,Z 423.072,A -85,B 0,C 180,E1 -10991.04,E2 -10991.04} C_VEL
LIN {X 0,Y 403.623,Z 427.135,A -85,B 0,C 180,E1 -10992.935,E2 -10992.935} C_VEL
LIN {X 0,Y 406.886,Z 440.506,A -85,B 0,C 180,E1 -10993.579,E2 -10993.579} C_VEL
LIN {X 0,Y 408.672,Z 450.72,A -85,B 0,C 180,E1 -10994.181,E2 -10994.181} C_VEL
LIN {X 0,Y 408.199,Z 461.494,A -85,B 0,C 180,E1 -10994.851,E2 -10994.851} C_VEL
LIN {X 0,Y 407.384,Z 473.154,A -85,B 0,C 180,E1 -10995.768,E2 -10995.768} C_VEL
LIN {X 0,Y 406.446,Z 485.018,A -85,B 0,C 180,E1 -10996.965,E2 -10996.965} C_VEL
LIN {X 0,Y 405.662,Z 494.633,A -85,B 0,C 180,E1 -10998.17,E2 -10998.17} C_VEL
LIN {X 0,Y 404.939,Z 503.331,A -85,B 0,C 180,E1 -10999.517,E2 -10999.517} C_VEL
LIN {X 0,Y 404.205,Z 511.831,A -85,B 0,C 180,E1 -11001.148,E2 -11001.148} C_VEL
LIN {X 0,Y 403.709,Z 518.132,A -85,B 0,C 180,E1 -11002.68,E2 -11002.68} C_VEL
LIN {X 0,Y 403.327,Z 522.99,A -85,B 0,C 180,E1 -11004.172,E2 -11004.172} C_VEL
LIN {X 0,Y 403.085,Z 527.1,A -85,B 0,C 180,E1 -11005.841,E2 -11005.841} C_VEL
LIN {X 0,Y 402.888,Z 529.489,A -85,B 0,C 180,E1 -11007.169,E2 -11007.169} C_VEL
LIN {X 0,Y 402.794,Z 530.706,A -85,B 0,C 180,E1 -11008.105,E2 -11008.105} C_VEL
LIN {X 0,Y 402.713,Z 531.734,A -85,B 0,C 180,E1 -11009.251,E2 -11009.251} C_VEL
LIN {X 0,Y 402.637,Z 532.208,A -85,B 0,C 180,E1 -11011.206,E2 -11011.206} C_VEL
LIN {X 0,Y 402.711,Z 531.218,A -85,B 0,C 180,E1 -11013.102,E2 -11013.102} C_VEL
LIN {X 0,Y 402.835,Z 528.886,A -85,B 0,C 180,E1 -11014.915,E2 -11014.915} C_VEL
LIN {X 0,Y 403.086,Z 525.243,A -85,B 0,C 180,E1 -11016.674,E2 -11016.674} C_VEL
LIN {X 0,Y 403.352,Z 520.39,A -85,B 0,C 180,E1 -11018.363,E2 -11018.363} C_VEL
LIN {X 0,Y 403.782,Z 513.823,A -85,B 0,C 180,E1 -11020.09,E2 -11020.09} C_VEL
LIN {X 0,Y 404.299,Z 506.387,A -85,B 0,C 180,E1 -11021.626,E2 -11021.626} C_VEL
LIN {X 0,Y 404.831,Z 498.675,A -85,B 0,C 180,E1 -11022.923,E2 -11022.923} C_VEL
LIN {X 0,Y 405.59,Z 489.268,A -85,B 0,C 180,E1 -11024.216,E2 -11024.216} C_VEL
LIN {X 0,Y 406.288,Z 479.12,A -85,B 0,C 180,E1 -11025.347,E2 -11025.347} C_VEL
LIN {X 0,Y 407.042,Z 467.456,A -85,B 0,C 180,E1 -11026.393,E2 -11026.393} C_VEL
LIN {X 0,Y 407.738,Z 456.121,A -85,B 0,C 180,E1 -11027.181,E2 -11027.181} C_VEL
LIN {X 0,Y 407.968,Z 449.897,A -85,B 0,C 180,E1 -11027.538,E2 -11027.538} C_VEL
LIN {X 0,Y 405.462,Z 436.274,A -85,B 0,C 180,E1 -11028.261,E2 -11028.261} C_VEL
LIN {X 0,Y 403.435,Z 426.16,A -85,B 0,C 180,E1 -11028.683,E2 -11028.683} C_VEL
LIN {X 0,Y 403.54,Z 420.283,A -85,B 0,C 180,E1 -11031.601,E2 -11031.601} C_VEL
LIN {X 0,Y 403.754,Z 413.564,A -85,B 0,C 180,E1 -11034.939,E2 -11034.939} C_VEL
LIN {X 0,Y 403.884,Z 407.528,A -85,B 0,C 180,E1 -11037.944,E2 -11037.944} C_VEL
LIN {X 0,Y 404.053,Z 400.555,A -85,B 0,C 180,E1 -11041.422,E2 -11041.422} C_VEL
LIN {X 0,Y 404.29,Z 392.686,A -85,B 0,C 180,E1 -11045.34,E2 -11045.34} C_VEL
LIN {X 0,Y 404.277,Z 390.129,A -85,B 0,C 180,E1 -11046.638,E2 -11046.638} C_VEL
LIN {X 0,Y 404.194,Z 390.137,A -85,B 0,C 180,E1 -11049.873,E2 -11049.873} C_VEL
LIN {X 0,Y 404.218,Z 390.134,A -85,B 0,C 180,E1 -11052.991,E2 -11052.991} C_VEL
LIN {X 0,Y 404.284,Z 390.128,A -85,B 0,C 180,E1 -11056.937,E2 -11056.937} C_VEL
LIN {X 0,Y 404.258,Z 390.132,A -85,B 0,C 180,E1 -11059.986,E2 -11059.986} C_VEL
LIN {X 0,Y 404.369,Z 390.118,A -85,B 0,C 180,E1 -11063.01,E2 -11063.01} C_VEL
LIN {X 0,Y 404.268,Z 390.132,A -85,B 0,C 180,E1 -11065.011,E2 -11065.011} C_VEL
LIN {X 0,Y 404.456,Z 390.107,A -85,B 0,C 180,E1 -11068.504,E2 -11068.504} C_VEL
LIN {X 0,Y 404.5,Z 390.468,A -85,B 0,C 180,E1 -11069.002,E2 -11069.002} C_VEL
LIN {X 0,Y 404.744,Z 391.997,A -85,B 0,C 180,E1 -11069.998,E2 -11069.998} C_VEL
LIN {X 0,Y 404.35,Z 396.809,A -85,B 0,C 180,E1 -11072.987,E2 -11072.987} C_VEL
LIN {X 0,Y 404.159,Z 401.736,A -85,B 0,C 180,E1 -11075.986,E2 -11075.986} C_VEL
LIN {X 0,Y 403.902,Z 406.683,A -85,B 0,C 180,E1 -11078.956,E2 -11078.956} C_VEL
LIN {X 0,Y 403.213,Z 408.12,A -85,B 0,C 180,E1 -11079.762,E2 -11079.762} C_VEL
LIN {X 0,Y 400.287,Z 410.654,A -85,B 0,C 180,E1 -11081.062,E2 -11081.062} C_VEL
LIN {X 0,Y 397.782,Z 412.703,A -85,B 0,C 180,E1 -11082.111,E2 -11082.111} C_VEL
LIN {X 0,Y 396.662,Z 414.198,A -85,B 0,C 180,E1 -11082.926,E2 -11082.926} C_VEL
LIN {X 0,Y 396.547,Z 414.679,A -85,B 0,C 180,E1 -11083.203,E2 -11083.203} C_VEL
LIN {X 0,Y 396.284,Z 420.7,A -85,B 0,C 180,E1 -11086.73,E2 -11086.73} C_VEL
LIN {X 0,Y 396.218,Z 423.743,A -85,B 0,C 180,E1 -11088.382,E2 -11088.382} C_VEL
LIN {X 0,Y 398.43,Z 434.844,A -85,B 0,C 180,E1 -11088.909,E2 -11088.909} C_VEL
LIN {X 0,Y 399.904,Z 444.319,A -85,B 0,C 180,E1 -11089.503,E2 -11089.503} C_VEL
LIN {X 0,Y 399.361,Z 455.614,A -85,B 0,C 180,E1 -11090.335,E2 -11090.335} C_VEL
LIN {X 0,Y 398.708,Z 465.523,A -85,B 0,C 180,E1 -11091.294,E2 -11091.294} C_VEL
LIN {X 0,Y 398.129,Z 473.854,A -85,B 0,C 180,E1 -11092.302,E2 -11092.302} C_VEL
LIN {X 0,Y 397.527,Z 482.183,A -85,B 0,C 180,E1 -11093.568,E2 -11093.568} C_VEL
LIN {X 0,Y 397.036,Z 488.971,A -85,B 0,C 180,E1 -11094.857,E2 -11094.857} C_VEL
LIN {X 0,Y 396.615,Z 494.886,A -85,B 0,C 180,E1 -11096.292,E2 -11096.292} C_VEL
LIN {X 0,Y 396.251,Z 500.272,A -85,B 0,C 180,E1 -11098.038,E2 -11098.038} C_VEL
LIN {X 0,Y 396.021,Z 503.952,A -85,B 0,C 180,E1 -11099.792,E2 -11099.792} C_VEL
LIN {X 0,Y 395.807,Z 506.042,A -85,B 0,C 180,E1 -11101.539,E2 -11101.539} C_VEL
LIN {X 0,Y 395.78,Z 506.678,A -85,B 0,C 180,E1 -11103.427,E2 -11103.427} C_VEL
LIN {X 0,Y 395.909,Z 505.704,A -85,B 0,C 180,E1 -11105.258,E2 -11105.258} C_VEL
LIN {X 0,Y 396.163,Z 503.103,A -85,B 0,C 180,E1 -11107.093,E2 -11107.093} C_VEL
LIN {X 0,Y 396.488,Z 499.236,A -85,B 0,C 180,E1 -11108.747,E2 -11108.747} C_VEL
LIN {X 0,Y 396.829,Z 495.2,A -85,B 0,C 180,E1 -11110.02,E2 -11110.02} C_VEL
LIN {X 0,Y 397.28,Z 489.282,A -85,B 0,C 180,E1 -11111.475,E2 -11111.475} C_VEL
LIN {X 0,Y 397.84,Z 482.09,A -85,B 0,C 180,E1 -11112.848,E2 -11112.848} C_VEL
LIN {X 0,Y 398.443,Z 474.501,A -85,B 0,C 180,E1 -11114.009,E2 -11114.009} C_VEL
LIN {X 0,Y 399.273,Z 464.204,A -85,B 0,C 180,E1 -11115.245,E2 -11115.245} C_VEL
LIN {X 0,Y 399.973,Z 453.803,A -85,B 0,C 180,E1 -11116.206,E2 -11116.206} C_VEL
LIN {X 0,Y 400.482,Z 445.439,A -85,B 0,C 180,E1 -11116.812,E2 -11116.812} C_VEL
LIN {X 0,Y 398.575,Z 434.12,A -85,B 0,C 180,E1 -11117.546,E2 -11117.546} C_VEL
LIN {X 0,Y 396.365,Z 424.131,A -85,B 0,C 180,E1 -11118.067,E2 -11118.067} C_VEL
LIN {X 0,Y 396.54,Z 418.126,A -85,B 0,C 180,E1 -11121.661,E2 -11121.661} C_VEL
LIN {X 0,Y 396.739,Z 413.354,A -85,B 0,C 180,E1 -11124.568,E2 -11124.568} C_VEL
LIN {X 0,Y 396.989,Z 407.496,A -85,B 0,C 180,E1 -11128.179,E2 -11128.179} C_VEL
LIN {X 0,Y 397.297,Z 402.309,A -85,B 0,C 180,E1 -11131.47,E2 -11131.47} C_VEL
LIN {X 0,Y 397.6,Z 396.93,A -85,B 0,C 180,E1 -11134.899,E2 -11134.899} C_VEL
LIN {X 0,Y 397.515,Z 393.633,A -85,B 0,C 180,E1 -11137.111,E2 -11137.111} C_VEL
LIN {X 0,Y 397.16,Z 391.016,A -85,B 0,C 180,E1 -11139.002,E2 -11139.002} C_VEL
LIN {X 0,Y 397.158,Z 391.019,A -85,B 0,C 180,E1 -11142.844,E2 -11142.844} C_VEL
LIN {X 0,Y 397.202,Z 391.01,A -85,B 0,C 180,E1 -11146.679,E2 -11146.679} C_VEL
LIN {X 0,Y 397.209,Z 391.009,A -85,B 0,C 180,E1 -11149.809,E2 -11149.809} C_VEL
LIN {X 0,Y 397.341,Z 390.994,A -85,B 0,C 180,E1 -11152.888,E2 -11152.888} C_VEL
LIN {X 0,Y 397.241,Z 391.005,A -85,B 0,C 180,E1 -11154.925,E2 -11154.925} C_VEL
LIN {X 0,Y 397.43,Z 390.98,A -85,B 0,C 180,E1 -11157.974,E2 -11157.974} C_VEL
LIN {X 0,Y 397.56,Z 390.964,A -85,B 0,C 180,E1 -11160,E2 -11160} C_VEL
LIN {X 0,Y 397.367,Z 390.989,A -85,B 0,C 180,E1 -11163.042,E2 -11163.042} C_VEL
LIN {X 0,Y 397.365,Z 390.986,A -85,B 0,C 180,E1 -11166.092,E2 -11166.092} C_VEL
LIN {X 0,Y 397.354,Z 390.99,A -85,B 0,C 180,E1 -11168.135,E2 -11168.135} C_VEL
LIN {X 0,Y 397.21,Z 391.005,A -85,B 0,C 180,E1 -11172.259,E2 -11172.259} C_VEL
LIN {X 0,Y 397.164,Z 391.01,A -85,B 0,C 180,E1 -11175.393,E2 -11175.393} C_VEL
LIN {X 0,Y 397.152,Z 391.011,A -85,B 0,C 180,E1 -11178.574,E2 -11178.574} C_VEL
LIN {X 0,Y 397.139,Z 391.013,A -85,B 0,C 180,E1 -11181.816,E2 -11181.816} C_VEL
LIN {X 0,Y 397.132,Z 391.017,A -85,B 0,C 180,E1 -11185.514,E2 -11185.514} C_VEL
LIN {X 0,Y 397.108,Z 391.021,A -85,B 0,C 180,E1 -11188.545,E2 -11188.545} C_VEL
LIN {X 0,Y 397.062,Z 391.023,A -85,B 0,C 180,E1 -11192.073,E2 -11192.073} C_VEL
LIN {X 0,Y 397.103,Z 391.022,A -85,B 0,C 180,E1 -11195.506,E2 -11195.506} C_VEL
LIN {X 0,Y 397.121,Z 391.019,A -85,B 0,C 180,E1 -11198.865,E2 -11198.865} C_VEL
LIN {X 0,Y 397.145,Z 391.018,A -85,B 0,C 180,E1 -11202.258,E2 -11202.258} C_VEL
LIN {X 0,Y 397.138,Z 391.015,A -85,B 0,C 180,E1 -11205.062,E2 -11205.062} C_VEL
LIN {X 0,Y 397.144,Z 391.017,A -85,B 0,C 180,E1 -11208.009,E2 -11208.009} C_VEL
LIN {X 0,Y 397.126,Z 391.128,A -85,B 0,C 180,E1 -11211.14,E2 -11211.14} C_VEL
LIN {X 0,Y 398.549,Z 398.049,A -85,B 0,C 180,E1 -11214.418,E2 -11214.418} C_VEL
LIN {X 0,Y 399.628,Z 403.819,A -85,B 0,C 180,E1 -11216.967,E2 -11216.967} C_VEL
LIN {X 0,Y 400.252,Z 408.292,A -85,B 0,C 180,E1 -11218.807,E2 -11218.807} C_VEL
LIN {X 0,Y 399.476,Z 415.655,A -85,B 0,C 180,E1 -11221.601,E2 -11221.601} C_VEL
LIN {X 0,Y 398.392,Z 426.469,A -85,B 0,C 180,E1 -11225.511,E2 -11225.511} C_VEL
LIN {X 0,Y 397.478,Z 437.358,A -85,B 0,C 180,E1 -11229.293,E2 -11229.293} C_VEL
LIN {X 0,Y 396.911,Z 445.918,A -85,B 0,C 180,E1 -11232.154,E2 -11232.154} C_VEL
LIN {X 0,Y 399.113,Z 459.255,A -85,B 0,C 180,E1 -11232.652,E2 -11232.652} C_VEL
LIN {X 0,Y 400.366,Z 472.032,A -85,B 0,C 180,E1 -11233.31,E2 -11233.31} C_VEL
LIN {X 0,Y 400.364,Z 479.31,A -85,B 0,C 180,E1 -11233.756,E2 -11233.756} C_VEL
LIN {X 0,Y 399.555,Z 490.47,A -85,B 0,C 180,E1 -11234.574,E2 -11234.574} C_VEL
LIN {X 0,Y 398.701,Z 501.225,A -85,B 0,C 180,E1 -11235.585,E2 -11235.585} C_VEL
LIN {X 0,Y 398.004,Z 510.991,A -85,B 0,C 180,E1 -11236.732,E2 -11236.732} C_VEL
LIN {X 0,Y 397.298,Z 521.61,A -85,B 0,C 180,E1 -11238.265,E2 -11238.265} C_VEL
LIN {X 0,Y 396.703,Z 528.935,A -85,B 0,C 180,E1 -11239.54,E2 -11239.54} C_VEL
LIN {X 0,Y 396.312,Z 536.119,A -85,B 0,C 180,E1 -11241.076,E2 -11241.076} C_VEL
LIN {X 0,Y 396.056,Z 540.954,A -85,B 0,C 180,E1 -11242.354,E2 -11242.354} C_VEL
LIN {X 0,Y 395.816,Z 546.421,A -85,B 0,C 180,E1 -11244.212,E2 -11244.212} C_VEL
LIN {X 0,Y 395.798,Z 550.034,A -85,B 0,C 180,E1 -11245.929,E2 -11245.929} C_VEL
LIN {X 0,Y 395.759,Z 551.59,A -85,B 0,C 180,E1 -11246.948,E2 -11246.948} C_VEL
LIN {X 0,Y 395.843,Z 552.682,A -85,B 0,C 180,E1 -11247.967,E2 -11247.967} C_VEL
LIN {X 0,Y 395.835,Z 553.351,A -85,B 0,C 180,E1 -11248.985,E2 -11248.985} C_VEL
LIN {X 0,Y 395.799,Z 553.62,A -85,B 0,C 180,E1 -11250.002,E2 -11250.002} C_VEL
LIN {X 0,Y 395.836,Z 553.479,A -85,B 0,C 180,E1 -11251.02,E2 -11251.02} C_VEL
LIN {X 0,Y 395.851,Z 552.886,A -85,B 0,C 180,E1 -11252.037,E2 -11252.037} C_VEL
LIN {X 0,Y 395.8,Z 550.487,A -85,B 0,C 180,E1 -11254.075,E2 -11254.075} C_VEL
LIN {X 0,Y 395.838,Z 547.028,A -85,B 0,C 180,E1 -11255.819,E2 -11255.819} C_VEL
LIN {X 0,Y 396.066,Z 541.893,A -85,B 0,C 180,E1 -11257.65,E2 -11257.65} C_VEL
LIN {X 0,Y 396.414,Z 536.283,A -85,B 0,C 180,E1 -11259.183,E2 -11259.183} C_VEL
LIN {X 0,Y 396.856,Z 529.276,A -85,B 0,C 180,E1 -11260.718,E2 -11260.718} C_VEL
LIN {X 0,Y 397.641,Z 520.506,A -85,B 0,C 180,E1 -11262.247,E2 -11262.247} C_VEL
LIN {X 0,Y 398.369,Z 510.693,A -85,B 0,C 180,E1 -11263.634,E2 -11263.634} C_VEL
LIN {X 0,Y 399.209,Z 500.458,A -85,B 0,C 180,E1 -11264.792,E2 -11264.792} C_VEL
LIN {X 0,Y 400.126,Z 489.335,A -85,B 0,C 180,E1 -11265.8,E2 -11265.8} C_VEL
LIN {X 0,Y 400.946,Z 477.554,A -85,B 0,C 180,E1 -11266.643,E2 -11266.643} C_VEL
LIN {X 0,Y 400.589,Z 468.615,A -85,B 0,C 180,E1 -11267.185,E2 -11267.185} C_VEL
LIN {X 0,Y 399.269,Z 456.746,A -85,B 0,C 180,E1 -11267.795,E2 -11267.795} C_VEL
LIN {X 0,Y 396.95,Z 444.156,A -85,B 0,C 180,E1 -11268.319,E2 -11268.319} C_VEL
LIN {X 0,Y 397.65,Z 433.854,A -85,B 0,C 180,E1 -11271.788,E2 -11271.788} C_VEL
LIN {X 0,Y 398.562,Z 423.085,A -85,B 0,C 180,E1 -11275.506,E2 -11275.506} C_VEL
LIN {X 0,Y 399.561,Z 413.433,A -85,B 0,C 180,E1 -11278.929,E2 -11278.929} C_VEL
LIN {X 0,Y 400.075,Z 407.171,A -85,B 0,C 180,E1 -11281.215,E2 -11281.215} C_VEL
LIN {X 0,Y 399.083,Z 401.214,A -85,B 0,C 180,E1 -11283.58,E2 -11283.58} C_VEL
LIN {X 0,Y 397.516,Z 393.116,A -85,B 0,C 180,E1 -11286.951,E2 -11286.951} C_VEL
LIN {X 0,Y 397.103,Z 391.022,A -85,B 0,C 180,E1 -11287.858,E2 -11287.858} C_VEL
LIN {X 0,Y 397.053,Z 391.026,A -85,B 0,C 180,E1 -11290.915,E2 -11290.915} C_VEL
LIN {X 0,Y 397.093,Z 391.024,A -85,B 0,C 180,E1 -11293.651,E2 -11293.651} C_VEL
LIN {X 0,Y 397.098,Z 391.015,A -85,B 0,C 180,E1 -11296.523,E2 -11296.523} C_VEL
LIN {X 0,Y 397.093,Z 391.021,A -85,B 0,C 180,E1 -11300.42,E2 -11300.42} C_VEL
LIN {X 0,Y 397.104,Z 391.02,A -85,B 0,C 180,E1 -11303.005,E2 -11303.005} C_VEL
LIN {X 0,Y 397.105,Z 391.023,A -85,B 0,C 180,E1 -11306.287,E2 -11306.287} C_VEL
LIN {X 0,Y 397.083,Z 391.021,A -85,B 0,C 180,E1 -11309.118,E2 -11309.118} C_VEL
LIN {X 0,Y 397.065,Z 391.024,A -85,B 0,C 180,E1 -11312.253,E2 -11312.253} C_VEL
LIN {X 0,Y 397.108,Z 391.021,A -85,B 0,C 180,E1 -11314.865,E2 -11314.865} C_VEL
LIN {X 0,Y 397.101,Z 391.021,A -85,B 0,C 180,E1 -11318.181,E2 -11318.181} C_VEL
LIN {X 0,Y 397.169,Z 391.012,A -85,B 0,C 180,E1 -11321.427,E2 -11321.427} C_VEL
LIN {X 0,Y 397.185,Z 391.013,A -85,B 0,C 180,E1 -11324.608,E2 -11324.608} C_VEL
LIN {X 0,Y 397.223,Z 391.007,A -85,B 0,C 180,E1 -11327.742,E2 -11327.742} C_VEL
LIN {X 0,Y 397.234,Z 391.005,A -85,B 0,C 180,E1 -11330.837,E2 -11330.837} C_VEL
LIN {X 0,Y 397.325,Z 390.995,A -85,B 0,C 180,E1 -11333.907,E2 -11333.907} C_VEL
LIN {X 0,Y 397.227,Z 391.013,A -85,B 0,C 180,E1 -11334.924,E2 -11334.924} C_VEL
LIN {X 0,Y 397.548,Z 395.192,A -85,B 0,C 180,E1 -11336.96,E2 -11336.96} C_VEL
LIN {X 0,Y 397.529,Z 400.44,A -85,B 0,C 180,E1 -11339.493,E2 -11339.493} C_VEL
LIN {X 0,Y 397.047,Z 407.777,A -85,B 0,C 180,E1 -11343.044,E2 -11343.044} C_VEL
LIN {X 0,Y 397.032,Z 413.041,A -85,B 0,C 180,E1 -11345.587,E2 -11345.587} C_VEL
LIN {X 0,Y 396.841,Z 419.255,A -85,B 0,C 180,E1 -11348.658,E2 -11348.658} C_VEL
LIN {X 0,Y 396.62,Z 427.091,A -85,B 0,C 180,E1 -11352.533,E2 -11352.533} C_VEL
LIN {X 0,Y 400.165,Z 441.766,A -85,B 0,C 180,E1 -11353.278,E2 -11353.278} C_VEL
LIN {X 0,Y 402.011,Z 453.041,A -85,B 0,C 180,E1 -11353.973,E2 -11353.973} C_VEL
LIN {X 0,Y 401.254,Z 464.602,A -85,B 0,C 180,E1 -11354.741,E2 -11354.741} C_VEL
LIN {X 0,Y 400.404,Z 476.246,A -85,B 0,C 180,E1 -11355.734,E2 -11355.734} C_VEL
LIN {X 0,Y 399.474,Z 486.915,A -85,B 0,C 180,E1 -11356.875,E2 -11356.875} C_VEL
LIN {X 0,Y 398.672,Z 496.165,A -85,B 0,C 180,E1 -11358.102,E2 -11358.102} C_VEL
LIN {X 0,Y 397.826,Z 505.416,A -85,B 0,C 180,E1 -11359.612,E2 -11359.612} C_VEL
LIN {X 0,Y 397.201,Z 512.275,A -85,B 0,C 180,E1 -11360.995,E2 -11360.995} C_VEL
LIN {X 0,Y 396.714,Z 517.761,A -85,B 0,C 180,E1 -11362.34,E2 -11362.34} C_VEL
LIN {X 0,Y 396.278,Z 523.339,A -85,B 0,C 180,E1 -11364.073,E2 -11364.073} C_VEL
LIN {X 0,Y 396.025,Z 527.411,A -85,B 0,C 180,E1 -11365.771,E2 -11365.771} C_VEL
LIN {X 0,Y 395.763,Z 530.286,A -85,B 0,C 180,E1 -11367.497,E2 -11367.497} C_VEL
LIN {X 0,Y 395.61,Z 532.089,A -85,B 0,C 180,E1 -11369.483,E2 -11369.483} C_VEL
LIN {X 0,Y 395.566,Z 532.346,A -85,B 0,C 180,E1 -11371.479,E2 -11371.479} C_VEL
LIN {X 0,Y 395.622,Z 531.109,A -85,B 0,C 180,E1 -11373.414,E2 -11373.414} C_VEL
LIN {X 0,Y 395.8,Z 528.568,A -85,B 0,C 180,E1 -11375.233,E2 -11375.233} C_VEL
LIN {X 0,Y 396.082,Z 524.52,A -85,B 0,C 180,E1 -11377.105,E2 -11377.105} C_VEL
LIN {X 0,Y 396.341,Z 519.695,A -85,B 0,C 180,E1 -11378.718,E2 -11378.718} C_VEL
LIN {X 0,Y 396.788,Z 513.217,A -85,B 0,C 180,E1 -11380.39,E2 -11380.39} C_VEL
LIN {X 0,Y 397.391,Z 505.195,A -85,B 0,C 180,E1 -11382.029,E2 -11382.029} C_VEL
LIN {X 0,Y 398.086,Z 496.016,A -85,B 0,C 180,E1 -11383.513,E2 -11383.513} C_VEL
LIN {X 0,Y 398.841,Z 486.077,A -85,B 0,C 180,E1 -11384.816,E2 -11384.816} C_VEL
LIN {X 0,Y 399.664,Z 474.756,A -85,B 0,C 180,E1 -11385.998,E2 -11385.998} C_VEL
LIN {X 0,Y 400.438,Z 463.156,A -85,B 0,C 180,E1 -11386.959,E2 -11386.959} C_VEL
LIN {X 0,Y 401.123,Z 451.787,A -85,B 0,C 180,E1 -11387.689,E2 -11387.689} C_VEL
LIN {X 0,Y 398.968,Z 439.308,A -85,B 0,C 180,E1 -11388.39,E2 -11388.39} C_VEL
LIN {X 0,Y 396.348,Z 426.323,A -85,B 0,C 180,E1 -11388.956,E2 -11388.956} C_VEL
LIN {X 0,Y 396.528,Z 419.647,A -85,B 0,C 180,E1 -11392.303,E2 -11392.303} C_VEL
LIN {X 0,Y 396.746,Z 413.329,A -85,B 0,C 180,E1 -11395.467,E2 -11395.467} C_VEL
LIN {X 0,Y 396.906,Z 406.104,A -85,B 0,C 180,E1 -11399.101,E2 -11399.101} C_VEL
LIN {X 0,Y 397.097,Z 399.144,A -85,B 0,C 180,E1 -11402.601,E2 -11402.601} C_VEL
LIN {X 0,Y 397.354,Z 392.414,A -85,B 0,C 180,E1 -11405.994,E2 -11405.994} C_VEL
LIN {X 0,Y 397.238,Z 391.006,A -85,B 0,C 180,E1 -11406.725,E2 -11406.725} C_VEL
LIN {X 0,Y 397.15,Z 391.018,A -85,B 0,C 180,E1 -11410.351,E2 -11410.351} C_VEL
LIN {X 0,Y 397.168,Z 391.014,A -85,B 0,C 180,E1 -11413.551,E2 -11413.551} C_VEL
LIN {X 0,Y 397.23,Z 391.007,A -85,B 0,C 180,E1 -11416.701,E2 -11416.701} C_VEL
LIN {X 0,Y 397.218,Z 391.009,A -85,B 0,C 180,E1 -11419.807,E2 -11419.807} C_VEL
LIN {X 0,Y 397.318,Z 390.996,A -85,B 0,C 180,E1 -11422.885,E2 -11422.885} C_VEL
LIN {X 0,Y 397.24,Z 391.008,A -85,B 0,C 180,E1 -11424.923,E2 -11424.923} C_VEL
LIN {X 0,Y 397.415,Z 391.01,A -85,B 0,C 180,E1 -11428.636,E2 -11428.636} C_VEL
LIN {X 0,Y 397.719,Z 393.065,A -85,B 0,C 180,E1 -11429.998,E2 -11429.998} C_VEL
LIN {X 0,Y 397.316,Z 397.923,A -85,B 0,C 180,E1 -11433.04,E2 -11433.04} C_VEL
LIN {X 0,Y 397.114,Z 402.847,A -85,B 0,C 180,E1 -11436.093,E2 -11436.093} C_VEL
LIN {X 0,Y 396.836,Z 407.89,A -85,B 0,C 180,E1 -11439.169,E2 -11439.169} C_VEL
LIN {X 0,Y 396.586,Z 414.205,A -85,B 0,C 180,E1 -11442.925,E2 -11442.925} C_VEL
LIN {X 0,Y 396.547,Z 414.679,A -85,B 0,C 180,E1 -11443.203,E2 -11443.203} C_VEL
LIN {X 0,Y 395.792,Z 416.149,A -85,B 0,C 180,E1 -11444.023,E2 -11444.023} C_VEL
LIN {X 0,Y 392.815,Z 418.711,A -85,B 0,C 180,E1 -11445.345,E2 -11445.345} C_VEL
LIN {X 0,Y 390.323,Z 420.773,A -85,B 0,C 180,E1 -11446.413,E2 -11446.413} C_VEL
LIN {X 0,Y 389.242,Z 422.281,A -85,B 0,C 180,E1 -11447.243,E2 -11447.243} C_VEL
LIN {X 0,Y 389.146,Z 422.767,A -85,B 0,C 180,E1 -11447.526,E2 -11447.526} C_VEL
LIN {X 0,Y 389.13,Z 423.709,A -85,B 0,C 180,E1 -11448.082,E2 -11448.082} C_VEL
LIN {X 0,Y 391.599,Z 436.138,A -85,B 0,C 180,E1 -11448.709,E2 -11448.709} C_VEL
LIN {X 0,Y 392.992,Z 445.463,A -85,B 0,C 180,E1 -11449.317,E2 -11449.317} C_VEL
LIN {X 0,Y 392.421,Z 456.542,A -85,B 0,C 180,E1 -11450.164,E2 -11450.164} C_VEL
LIN {X 0,Y 391.737,Z 466.06,A -85,B 0,C 180,E1 -11451.108,E2 -11451.108} C_VEL
LIN {X 0,Y 391.144,Z 474.579,A -85,B 0,C 180,E1 -11452.165,E2 -11452.165} C_VEL
LIN {X 0,Y 390.478,Z 483.537,A -85,B 0,C 180,E1 -11453.576,E2 -11453.576} C_VEL
LIN {X 0,Y 389.932,Z 490.807,A -85,B 0,C 180,E1 -11455.05,E2 -11455.05} C_VEL
LIN {X 0,Y 389.575,Z 495.434,A -85,B 0,C 180,E1 -11456.227,E2 -11456.227} C_VEL
LIN {X 0,Y 389.213,Z 500.207,A -85,B 0,C 180,E1 -11457.775,E2 -11457.775} C_VEL
LIN {X 0,Y 389.02,Z 503.373,A -85,B 0,C 180,E1 -11459.191,E2 -11459.191} C_VEL
LIN {X 0,Y 388.851,Z 505.297,A -85,B 0,C 180,E1 -11460.399,E2 -11460.399} C_VEL
LIN {X 0,Y 388.714,Z 506.665,A -85,B 0,C 180,E1 -11461.814,E2 -11461.814} C_VEL
LIN {X 0,Y 388.721,Z 507.051,A -85,B 0,C 180,E1 -11463.73,E2 -11463.73} C_VEL
LIN {X 0,Y 388.878,Z 505.829,A -85,B 0,C 180,E1 -11465.585,E2 -11465.585} C_VEL
LIN {X 0,Y 389.005,Z 504.52,A -85,B 0,C 180,E1 -11466.594,E2 -11466.594} C_VEL
LIN {X 0,Y 389.235,Z 502.138,A -85,B 0,C 180,E1 -11467.868,E2 -11467.868} C_VEL
LIN {X 0,Y 389.623,Z 497.886,A -85,B 0,C 180,E1 -11469.478,E2 -11469.478} C_VEL
LIN {X 0,Y 390.015,Z 493.224,A -85,B 0,C 180,E1 -11470.815,E2 -11470.815} C_VEL
LIN {X 0,Y 390.468,Z 487.509,A -85,B 0,C 180,E1 -11472.119,E2 -11472.119} C_VEL
LIN {X 0,Y 391.152,Z 479.292,A -85,B 0,C 180,E1 -11473.586,E2 -11473.586} C_VEL
LIN {X 0,Y 391.873,Z 471.133,A -85,B 0,C 180,E1 -11474.738,E2 -11474.738} C_VEL
LIN {X 0,Y 392.69,Z 460.734,A -85,B 0,C 180,E1 -11475.895,E2 -11475.895} C_VEL
LIN {X 0,Y 393.471,Z 449.544,A -85,B 0,C 180,E1 -11476.838,E2 -11476.838} C_VEL
LIN {X 0,Y 393.471,Z 445.302,A -85,B 0,C 180,E1 -11477.142,E2 -11477.142} C_VEL
LIN {X 0,Y 391.807,Z 435.56,A -85,B 0,C 180,E1 -11477.796,E2 -11477.796} C_VEL
LIN {X 0,Y 389.328,Z 424.372,A -85,B 0,C 180,E1 -11478.398,E2 -11478.398} C_VEL
LIN {X 0,Y 389.57,Z 417.595,A -85,B 0,C 180,E1 -11482.534,E2 -11482.534} C_VEL
LIN {X 0,Y 389.785,Z 411.944,A -85,B 0,C 180,E1 -11486.031,E2 -11486.031} C_VEL
LIN {X 0,Y 390.135,Z 405.968,A -85,B 0,C 180,E1 -11489.84,E2 -11489.84} C_VEL
LIN {X 0,Y 390.457,Z 400.617,A -85,B 0,C 180,E1 -11493.258,E2 -11493.258} C_VEL
LIN {X 0,Y 390.562,Z 397.162,A -85,B 0,C 180,E1 -11495.552,E2 -11495.552} C_VEL
LIN {X 0,Y 390.408,Z 393.942,A -85,B 0,C 180,E1 -11497.788,E2 -11497.788} C_VEL
LIN {X 0,Y 390.15,Z 391.889,A -85,B 0,C 180,E1 -11499.36,E2 -11499.36} C_VEL
LIN {X 0,Y 390.114,Z 391.897,A -85,B 0,C 180,E1 -11503.248,E2 -11503.248} C_VEL
LIN {X 0,Y 390.171,Z 391.886,A -85,B 0,C 180,E1 -11506.561,E2 -11506.561} C_VEL
LIN {X 0,Y 390.159,Z 391.888,A -85,B 0,C 180,E1 -11509.623,E2 -11509.623} C_VEL
LIN {X 0,Y 390.296,Z 391.872,A -85,B 0,C 180,E1 -11512.759,E2 -11512.759} C_VEL
LIN {X 0,Y 390.213,Z 391.88,A -85,B 0,C 180,E1 -11514.834,E2 -11514.834} C_VEL
LIN {X 0,Y 390.399,Z 391.856,A -85,B 0,C 180,E1 -11517.937,E2 -11517.937} C_VEL
LIN {X 0,Y 390.53,Z 391.84,A -85,B 0,C 180,E1 -11520,E2 -11520} C_VEL
LIN {X 0,Y 390.327,Z 391.865,A -85,B 0,C 180,E1 -11523.097,E2 -11523.097} C_VEL
LIN {X 0,Y 390.318,Z 391.863,A -85,B 0,C 180,E1 -11526.202,E2 -11526.202} C_VEL
LIN {X 0,Y 390.292,Z 391.87,A -85,B 0,C 180,E1 -11528.283,E2 -11528.283} C_VEL
LIN {X 0,Y 390.158,Z 391.883,A -85,B 0,C 180,E1 -11532.484,E2 -11532.484} C_VEL
LIN {X 0,Y 390.123,Z 391.887,A -85,B 0,C 180,E1 -11535.678,E2 -11535.678} C_VEL
LIN {X 0,Y 390.099,Z 391.889,A -85,B 0,C 180,E1 -11538.923,E2 -11538.923} C_VEL
LIN {X 0,Y 390.063,Z 391.898,A -85,B 0,C 180,E1 -11542.233,E2 -11542.233} C_VEL
LIN {X 0,Y 390.099,Z 391.894,A -85,B 0,C 180,E1 -11545.745,E2 -11545.745} C_VEL
LIN {X 0,Y 390.046,Z 391.898,A -85,B 0,C 180,E1 -11549.111,E2 -11549.111} C_VEL
LIN {X 0,Y 390.025,Z 391.9,A -85,B 0,C 180,E1 -11552.724,E2 -11552.724} C_VEL
LIN {X 0,Y 390.04,Z 391.901,A -85,B 0,C 180,E1 -11555.828,E2 -11555.828} C_VEL
LIN {X 0,Y 390.059,Z 391.9,A -85,B 0,C 180,E1 -11559.222,E2 -11559.222} C_VEL
LIN {X 0,Y 390.108,Z 391.894,A -85,B 0,C 180,E1 -11562.389,E2 -11562.389} C_VEL
LIN {X 0,Y 390.105,Z 391.89,A -85,B 0,C 180,E1 -11565.368,E2 -11565.368} C_VEL
LIN {X 0,Y 390.093,Z 391.894,A -85,B 0,C 180,E1 -11568.199,E2 -11568.199} C_VEL
LIN {X 0,Y 390.078,Z 391.965,A -85,B 0,C 180,E1 -11570.629,E2 -11570.629} C_VEL
LIN {X 0,Y 391.664,Z 399.794,A -85,B 0,C 180,E1 -11574.445,E2 -11574.445} C_VEL
LIN {X 0,Y 392.837,Z 406.028,A -85,B 0,C 180,E1 -11577.23,E2 -11577.23} C_VEL
LIN {X 0,Y 393.312,Z 409.765,A -85,B 0,C 180,E1 -11578.792,E2 -11578.792} C_VEL
LIN {X 0,Y 392.582,Z 416.287,A -85,B 0,C 180,E1 -11581.307,E2 -11581.307} C_VEL
LIN {X 0,Y 391.505,Z 426.338,A -85,B 0,C 180,E1 -11585.051,E2 -11585.051} C_VEL
LIN {X 0,Y 390.498,Z 437.152,A -85,B 0,C 180,E1 -11588.906,E2 -11588.906} C_VEL
LIN {X 0,Y 389.917,Z 445.645,A -85,B 0,C 180,E1 -11591.822,E2 -11591.822} C_VEL
LIN {X 0,Y 392.177,Z 459.297,A -85,B 0,C 180,E1 -11592.348,E2 -11592.348} C_VEL
LIN {X 0,Y 393.479,Z 472.361,A -85,B 0,C 180,E1 -11593.047,E2 -11593.047} C_VEL
LIN {X 0,Y 393.474,Z 479.967,A -85,B 0,C 180,E1 -11593.531,E2 -11593.531} C_VEL
LIN {X 0,Y 392.571,Z 491.576,A -85,B 0,C 180,E1 -11594.426,E2 -11594.426} C_VEL
LIN {X 0,Y 391.705,Z 502.045,A -85,B 0,C 180,E1 -11595.455,E2 -11595.455} C_VEL
LIN {X 0,Y 390.89,Z 512.585,A -85,B 0,C 180,E1 -11596.75,E2 -11596.75} C_VEL
LIN {X 0,Y 390.177,Z 522.796,A -85,B 0,C 180,E1 -11598.311,E2 -11598.311} C_VEL
LIN {X 0,Y 389.539,Z 531.124,A -85,B 0,C 180,E1 -11599.871,E2 -11599.871} C_VEL
LIN {X 0,Y 389.147,Z 537.817,A -85,B 0,C 180,E1 -11601.434,E2 -11601.434} C_VEL
LIN {X 0,Y 388.825,Z 543.883,A -85,B 0,C 180,E1 -11603.255,E2 -11603.255} C_VEL
LIN {X 0,Y 388.746,Z 547.787,A -85,B 0,C 180,E1 -11604.816,E2 -11604.816} C_VEL
LIN {X 0,Y 388.72,Z 549.783,A -85,B 0,C 180,E1 -11605.855,E2 -11605.855} C_VEL
LIN {X 0,Y 388.664,Z 551.35,A -85,B 0,C 180,E1 -11606.893,E2 -11606.893} C_VEL
LIN {X 0,Y 388.739,Z 552.464,A -85,B 0,C 180,E1 -11607.93,E2 -11607.93} C_VEL
LIN {X 0,Y 388.763,Z 553.144,A -85,B 0,C 180,E1 -11608.966,E2 -11608.966} C_VEL
LIN {X 0,Y 388.728,Z 553.422,A -85,B 0,C 180,E1 -11610.002,E2 -11610.002} C_VEL
LIN {X 0,Y 388.765,Z 553.298,A -85,B 0,C 180,E1 -11611.038,E2 -11611.038} C_VEL
LIN {X 0,Y 388.745,Z 552.718,A -85,B 0,C 180,E1 -11612.074,E2 -11612.074} C_VEL
LIN {X 0,Y 388.723,Z 550.343,A -85,B 0,C 180,E1 -11614.149,E2 -11614.149} C_VEL
LIN {X 0,Y 388.74,Z 547.28,A -85,B 0,C 180,E1 -11615.77,E2 -11615.77} C_VEL
LIN {X 0,Y 388.936,Z 543.419,A -85,B 0,C 180,E1 -11617.269,E2 -11617.269} C_VEL
LIN {X 0,Y 389.322,Z 537.255,A -85,B 0,C 180,E1 -11619.09,E2 -11619.09} C_VEL
LIN {X 0,Y 389.768,Z 530.508,A -85,B 0,C 180,E1 -11620.653,E2 -11620.653} C_VEL
LIN {X 0,Y 390.549,Z 522.155,A -85,B 0,C 180,E1 -11622.209,E2 -11622.209} C_VEL
LIN {X 0,Y 391.359,Z 512.336,A -85,B 0,C 180,E1 -11623.669,E2 -11623.669} C_VEL
LIN {X 0,Y 392.22,Z 501.895,A -85,B 0,C 180,E1 -11624.928,E2 -11624.928} C_VEL
LIN {X 0,Y 393.186,Z 491.225,A -85,B 0,C 180,E1 -11625.953,E2 -11625.953} C_VEL
LIN {X 0,Y 394.085,Z 479.852,A -85,B 0,C 180,E1 -11626.819,E2 -11626.819} C_VEL
LIN {X 0,Y 394.199,Z 474.487,A -85,B 0,C 180,E1 -11627.171,E2 -11627.171} C_VEL
LIN {X 0,Y 393.124,Z 461.389,A -85,B 0,C 180,E1 -11627.935,E2 -11627.935} C_VEL
LIN {X 0,Y 390.76,Z 447.902,A -85,B 0,C 180,E1 -11628.554,E2 -11628.554} C_VEL
LIN {X 0,Y 389.96,Z 443.615,A -85,B 0,C 180,E1 -11628.727,E2 -11628.727} C_VEL
LIN {X 0,Y 390.699,Z 433.561,A -85,B 0,C 180,E1 -11632.197,E2 -11632.197} C_VEL
LIN {X 0,Y 391.519,Z 424.149,A -85,B 0,C 180,E1 -11635.521,E2 -11635.521} C_VEL
LIN {X 0,Y 392.718,Z 413.188,A -85,B 0,C 180,E1 -11639.483,E2 -11639.483} C_VEL
LIN {X 0,Y 393.117,Z 408.531,A -85,B 0,C 180,E1 -11641.23,E2 -11641.23} C_VEL
LIN {X 0,Y 392.093,Z 402.28,A -85,B 0,C 180,E1 -11643.758,E2 -11643.758} C_VEL
LIN {X 0,Y 390.607,Z 394.658,A -85,B 0,C 180,E1 -11646.997,E2 -11646.997} C_VEL
LIN {X 0,Y 390.075,Z 391.898,A -85,B 0,C 180,E1 -11648.269,E2 -11648.269} C_VEL
LIN {X 0,Y 390.021,Z 391.904,A -85,B 0,C 180,E1 -11651.816,E2 -11651.816} C_VEL
LIN {X 0,Y 390.047,Z 391.899,A -85,B 0,C 180,E1 -11655.354,E2 -11655.354} C_VEL
LIN {X 0,Y 390.022,Z 391.901,A -85,B 0,C 180,E1 -11658.185,E2 -11658.185} C_VEL
LIN {X 0,Y 390.065,Z 391.896,A -85,B 0,C 180,E1 -11660.904,E2 -11660.904} C_VEL
LIN {X 0,Y 390.089,Z 391.894,A -85,B 0,C 180,E1 -11664.793,E2 -11664.793} C_VEL
LIN {X 0,Y 390.029,Z 391.9,A -85,B 0,C 180,E1 -11668.496,E2 -11668.496} C_VEL
LIN {X 0,Y 390.022,Z 391.903,A -85,B 0,C 180,E1 -11672.003,E2 -11672.003} C_VEL
LIN {X 0,Y 390.048,Z 391.899,A -85,B 0,C 180,E1 -11675.517,E2 -11675.517} C_VEL
LIN {X 0,Y 390.062,Z 391.899,A -85,B 0,C 180,E1 -11678.878,E2 -11678.878} C_VEL
LIN {X 0,Y 390.135,Z 391.891,A -85,B 0,C 180,E1 -11682.167,E2 -11682.167} C_VEL
LIN {X 0,Y 390.15,Z 391.89,A -85,B 0,C 180,E1 -11685.392,E2 -11685.392} C_VEL
LIN {X 0,Y 390.148,Z 391.888,A -85,B 0,C 180,E1 -11688.571,E2 -11688.571} C_VEL
LIN {X 0,Y 390.262,Z 391.874,A -85,B 0,C 180,E1 -11692.086,E2 -11692.086} C_VEL
LIN {X 0,Y 390.248,Z 392.084,A -85,B 0,C 180,E1 -11694.704,E2 -11694.704} C_VEL
LIN {X 0,Y 390.598,Z 396.526,A -85,B 0,C 180,E1 -11696.905,E2 -11696.905} C_VEL
LIN {X 0,Y 390.553,Z 401.722,A -85,B 0,C 180,E1 -11699.484,E2 -11699.484} C_VEL
LIN {X 0,Y 390.051,Z 409.124,A -85,B 0,C 180,E1 -11703.098,E2 -11703.098} C_VEL
LIN {X 0,Y 390.009,Z 415.449,A -85,B 0,C 180,E1 -11706.207,E2 -11706.207} C_VEL
LIN {X 0,Y 389.748,Z 421.738,A -85,B 0,C 180,E1 -11709.339,E2 -11709.339} C_VEL
LIN {X 0,Y 389.616,Z 427.242,A -85,B 0,C 180,E1 -11712.104,E2 -11712.104} C_VEL
LIN {X 0,Y 393.348,Z 442.414,A -85,B 0,C 180,E1 -11712.923,E2 -11712.923} C_VEL
LIN {X 0,Y 395.206,Z 453.052,A -85,B 0,C 180,E1 -11713.611,E2 -11713.611} C_VEL
LIN {X 0,Y 394.516,Z 465.167,A -85,B 0,C 180,E1 -11714.442,E2 -11714.442} C_VEL
LIN {X 0,Y 393.658,Z 476.243,A -85,B 0,C 180,E1 -11715.403,E2 -11715.403} C_VEL
LIN {X 0,Y 392.726,Z 486.481,A -85,B 0,C 180,E1 -11716.504,E2 -11716.504} C_VEL
LIN {X 0,Y 391.838,Z 495.861,A -85,B 0,C 180,E1 -11717.752,E2 -11717.752} C_VEL
LIN {X 0,Y 391.023,Z 504.416,A -85,B 0,C 180,E1 -11719.148,E2 -11719.148} C_VEL
LIN {X 0,Y 390.236,Z 512.525,A -85,B 0,C 180,E1 -11720.782,E2 -11720.782} C_VEL
LIN {X 0,Y 389.576,Z 519.664,A -85,B 0,C 180,E1 -11722.637,E2 -11722.637} C_VEL
LIN {X 0,Y 389.069,Z 525.213,A -85,B 0,C 180,E1 -11724.548,E2 -11724.548} C_VEL
LIN {X 0,Y 388.827,Z 528.806,A -85,B 0,C 180,E1 -11726.284,E2 -11726.284} C_VEL
LIN {X 0,Y 388.605,Z 531.226,A -85,B 0,C 180,E1 -11728.048,E2 -11728.048} C_VEL
LIN {X 0,Y 388.484,Z 532.421,A -85,B 0,C 180,E1 -11729.729,E2 -11729.729} C_VEL
LIN {X 0,Y 388.468,Z 532.452,A -85,B 0,C 180,E1 -11731.753,E2 -11731.753} C_VEL
LIN {X 0,Y 388.55,Z 531.001,A -85,B 0,C 180,E1 -11733.689,E2 -11733.689} C_VEL
LIN {X 0,Y 388.74,Z 528.262,A -85,B 0,C 180,E1 -11735.554,E2 -11735.554} C_VEL
LIN {X 0,Y 389.015,Z 524.234,A -85,B 0,C 180,E1 -11737.351,E2 -11737.351} C_VEL
LIN {X 0,Y 389.362,Z 518.613,A -85,B 0,C 180,E1 -11739.179,E2 -11739.179} C_VEL
LIN {X 0,Y 389.819,Z 512.276,A -85,B 0,C 180,E1 -11740.779,E2 -11740.779} C_VEL
LIN {X 0,Y 390.342,Z 505.748,A -85,B 0,C 180,E1 -11742.114,E2 -11742.114} C_VEL
LIN {X 0,Y 391.042,Z 496.788,A -85,B 0,C 180,E1 -11743.605,E2 -11743.605} C_VEL
LIN {X 0,Y 391.844,Z 486.987,A -85,B 0,C 180,E1 -11744.928,E2 -11744.928} C_VEL
LIN {X 0,Y 392.653,Z 476.331,A -85,B 0,C 180,E1 -11746.089,E2 -11746.089} C_VEL
LIN {X 0,Y 393.438,Z 464.796,A -85,B 0,C 180,E1 -11747.086,E2 -11747.086} C_VEL
LIN {X 0,Y 394.191,Z 453.376,A -85,B 0,C 180,E1 -11747.858,E2 -11747.858} C_VEL
LIN {X 0,Y 392.713,Z 443.598,A -85,B 0,C 180,E1 -11748.448,E2 -11748.448} C_VEL
LIN {X 0,Y 390.222,Z 430.936,A -85,B 0,C 180,E1 -11749.059,E2 -11749.059} C_VEL
LIN {X 0,Y 389.319,Z 426.469,A -85,B 0,C 180,E1 -11749.241,E2 -11749.241} C_VEL
LIN {X 0,Y 389.467,Z 419.908,A -85,B 0,C 180,E1 -11752.559,E2 -11752.559} C_VEL
LIN {X 0,Y 389.725,Z 413.003,A -85,B 0,C 180,E1 -11756.05,E2 -11756.05} C_VEL
LIN {X 0,Y 389.898,Z 405.423,A -85,B 0,C 180,E1 -11759.906,E2 -11759.906} C_VEL
LIN {X 0,Y 390.065,Z 398.887,A -85,B 0,C 180,E1 -11763.226,E2 -11763.226} C_VEL
LIN {X 0,Y 390.318,Z 393.238,A -85,B 0,C 180,E1 -11766.099,E2 -11766.099} C_VEL
LIN {X 0,Y 390.185,Z 391.885,A -85,B 0,C 180,E1 -11766.841,E2 -11766.841} C_VEL
LIN {X 0,Y 390.106,Z 391.892,A -85,B 0,C 180,E1 -11769.981,E2 -11769.981} C_VEL
LIN {X 0,Y 390.14,Z 391.888,A -85,B 0,C 180,E1 -11773.246,E2 -11773.246} C_VEL
LIN {X 0,Y 390.196,Z 391.883,A -85,B 0,C 180,E1 -11776.56,E2 -11776.56} C_VEL
LIN {X 0,Y 390.204,Z 391.879,A -85,B 0,C 180,E1 -11780.669,E2 -11780.669} C_VEL
LIN {X 0,Y 390.298,Z 391.871,A -85,B 0,C 180,E1 -11783.795,E2 -11783.795} C_VEL
LIN {X 0,Y 390.395,Z 391.874,A -85,B 0,C 180,E1 -11788.483,E2 -11788.483} C_VEL
LIN {X 0,Y 390.695,Z 394.132,A -85,B 0,C 180,E1 -11789.998,E2 -11789.998} C_VEL
LIN {X 0,Y 390.256,Z 398.995,A -85,B 0,C 180,E1 -11793.095,E2 -11793.095} C_VEL
LIN {X 0,Y 390.071,Z 403.967,A -85,B 0,C 180,E1 -11796.204,E2 -11796.204} C_VEL
LIN {X 0,Y 389.785,Z 409.058,A -85,B 0,C 180,E1 -11799.336,E2 -11799.336} C_VEL
LIN {X 0,Y 389.503,Z 415.349,A -85,B 0,C 180,E1 -11803.148,E2 -11803.148} C_VEL
LIN {X 0,Y 389.206,Z 421.635,A -85,B 0,C 180,E1 -11806.857,E2 -11806.857} C_VEL
LIN {X 0,Y 389.146,Z 422.767,A -85,B 0,C 180,E1 -11807.526,E2 -11807.526} C_VEL
LIN {X 0,Y 389.107,Z 424.277,A -85,B 0,C 180,E1 -11807.878,E2 -11807.878} C_VEL
LIN {X 0,Y 389.036,Z 426.719,A -85,B 0,C 180,E1 -11808.118,E2 -11808.118} C_VEL
LIN {X 0,Y 388.323,Z 436.651,A -85,B 0,C 180,E1 -11808.606,E2 -11808.606} C_VEL
LIN {X 0,Y 386.379,Z 447.479,A -85,B 0,C 180,E1 -11809.186,E2 -11809.186} C_VEL
LIN {X 0,Y 385.837,Z 451.459,A -85,B 0,C 180,E1 -11809.483,E2 -11809.483} C_VEL
LIN {X 0,Y 385.08,Z 461.986,A -85,B 0,C 180,E1 -11810.421,E2 -11810.421} C_VEL
LIN {X 0,Y 384.466,Z 470.959,A -85,B 0,C 180,E1 -11811.441,E2 -11811.441} C_VEL
LIN {X 0,Y 383.849,Z 479.16,A -85,B 0,C 180,E1 -11812.609,E2 -11812.609} C_VEL
LIN {X 0,Y 383.224,Z 487.372,A -85,B 0,C 180,E1 -11814.079,E2 -11814.079} C_VEL
LIN {X 0,Y 382.733,Z 493.192,A -85,B 0,C 180,E1 -11815.404,E2 -11815.404} C_VEL
LIN {X 0,Y 382.325,Z 497.952,A -85,B 0,C 180,E1 -11816.764,E2 -11816.764} C_VEL
LIN {X 0,Y 382.044,Z 502.637,A -85,B 0,C 180,E1 -11818.57,E2 -11818.57} C_VEL
LIN {X 0,Y 381.8,Z 505.322,A -85,B 0,C 180,E1 -11820.1,E2 -11820.1} C_VEL
LIN {X 0,Y 381.676,Z 506.446,A -85,B 0,C 180,E1 -11821.033,E2 -11821.033} C_VEL
LIN {X 0,Y 381.605,Z 507.304,A -85,B 0,C 180,E1 -11822.279,E2 -11822.279} C_VEL
LIN {X 0,Y 381.665,Z 507.374,A -85,B 0,C 180,E1 -11824.042,E2 -11824.042} C_VEL
LIN {X 0,Y 381.855,Z 505.96,A -85,B 0,C 180,E1 -11825.923,E2 -11825.923} C_VEL
LIN {X 0,Y 382.137,Z 503.046,A -85,B 0,C 180,E1 -11827.738,E2 -11827.738} C_VEL
LIN {X 0,Y 382.454,Z 499.836,A -85,B 0,C 180,E1 -11829.091,E2 -11829.091} C_VEL
LIN {X 0,Y 382.899,Z 495.092,A -85,B 0,C 180,E1 -11830.601,E2 -11830.601} C_VEL
LIN {X 0,Y 383.373,Z 489.408,A -85,B 0,C 180,E1 -11831.995,E2 -11831.995} C_VEL
LIN {X 0,Y 384.001,Z 482.113,A -85,B 0,C 180,E1 -11833.414,E2 -11833.414} C_VEL
LIN {X 0,Y 384.748,Z 473.937,A -85,B 0,C 180,E1 -11834.666,E2 -11834.666} C_VEL
LIN {X 0,Y 385.6,Z 464.556,A -85,B 0,C 180,E1 -11835.81,E2 -11835.81} C_VEL
LIN {X 0,Y 386.423,Z 453.26,A -85,B 0,C 180,E1 -11836.872,E2 -11836.872} C_VEL
LIN {X 0,Y 386.681,Z 446.735,A -85,B 0,C 180,E1 -11837.363,E2 -11837.363} C_VEL
LIN {X 0,Y 384.852,Z 436.027,A -85,B 0,C 180,E1 -11838.112,E2 -11838.112} C_VEL
LIN {X 0,Y 382.277,Z 424.615,A -85,B 0,C 180,E1 -11838.751,E2 -11838.751} C_VEL
LIN {X 0,Y 382.531,Z 418.285,A -85,B 0,C 180,E1 -11842.679,E2 -11842.679} C_VEL
LIN {X 0,Y 382.745,Z 413.46,A -85,B 0,C 180,E1 -11845.714,E2 -11845.714} C_VEL
LIN {X 0,Y 383.081,Z 407.473,A -85,B 0,C 180,E1 -11849.565,E2 -11849.565} C_VEL
LIN {X 0,Y 383.397,Z 402.574,A -85,B 0,C 180,E1 -11852.725,E2 -11852.725} C_VEL
LIN {X 0,Y 383.563,Z 399.122,A -85,B 0,C 180,E1 -11855.076,E2 -11855.076} C_VEL
LIN {X 0,Y 383.491,Z 395.831,A -85,B 0,C 180,E1 -11857.366,E2 -11857.366} C_VEL
LIN {X 0,Y 383.088,Z 392.769,A -85,B 0,C 180,E1 -11859.601,E2 -11859.601} C_VEL
LIN {X 0,Y 383.081,Z 392.773,A -85,B 0,C 180,E1 -11862.931,E2 -11862.931} C_VEL
LIN {X 0,Y 383.102,Z 392.766,A -85,B 0,C 180,E1 -11866.463,E2 -11866.463} C_VEL
LIN {X 0,Y 383.121,Z 392.764,A -85,B 0,C 180,E1 -11869.43,E2 -11869.43} C_VEL
LIN {X 0,Y 383.25,Z 392.748,A -85,B 0,C 180,E1 -11872.625,E2 -11872.625} C_VEL
LIN {X 0,Y 383.185,Z 392.756,A -85,B 0,C 180,E1 -11874.739,E2 -11874.739} C_VEL
LIN {X 0,Y 383.368,Z 392.732,A -85,B 0,C 180,E1 -11877.899,E2 -11877.899} C_VEL
LIN {X 0,Y 383.499,Z 392.716,A -85,B 0,C 180,E1 -11880,E2 -11880} C_VEL
LIN {X 0,Y 383.261,Z 392.744,A -85,B 0,C 180,E1 -11883.154,E2 -11883.154} C_VEL
LIN {X 0,Y 383.273,Z 392.739,A -85,B 0,C 180,E1 -11886.317,E2 -11886.317} C_VEL
LIN {X 0,Y 383.238,Z 392.75,A -85,B 0,C 180,E1 -11888.437,E2 -11888.437} C_VEL
LIN {X 0,Y 383.09,Z 392.766,A -85,B 0,C 180,E1 -11891.643,E2 -11891.643} C_VEL
LIN {X 0,Y 383.093,Z 392.766,A -85,B 0,C 180,E1 -11894.883,E2 -11894.883} C_VEL
LIN {X 0,Y 383.074,Z 392.765,A -85,B 0,C 180,E1 -11898.173,E2 -11898.173} C_VEL
LIN {X 0,Y 383.013,Z 392.772,A -85,B 0,C 180,E1 -11901.53,E2 -11901.53} C_VEL
LIN {X 0,Y 383.032,Z 392.772,A -85,B 0,C 180,E1 -11904.962,E2 -11904.962} C_VEL
LIN {X 0,Y 383.03,Z 392.774,A -85,B 0,C 180,E1 -11908.494,E2 -11908.494} C_VEL
LIN {X 0,Y 382.992,Z 392.775,A -85,B 0,C 180,E1 -11912.152,E2 -11912.152} C_VEL
LIN {X 0,Y 383.001,Z 392.777,A -85,B 0,C 180,E1 -11914.67,E2 -11914.67} C_VEL
LIN {X 0,Y 382.987,Z 392.78,A -85,B 0,C 180,E1 -11917.907,E2 -11917.907} C_VEL
LIN {X 0,Y 383.032,Z 392.775,A -85,B 0,C 180,E1 -11921.342,E2 -11921.342} C_VEL
LIN {X 0,Y 383.057,Z 392.772,A -85,B 0,C 180,E1 -11924.317,E2 -11924.317} C_VEL
LIN {X 0,Y 383.062,Z 392.769,A -85,B 0,C 180,E1 -11927.252,E2 -11927.252} C_VEL
LIN {X 0,Y 383.051,Z 392.945,A -85,B 0,C 180,E1 -11930.164,E2 -11930.164} C_VEL
LIN {X 0,Y 384.381,Z 399.685,A -85,B 0,C 180,E1 -11933.562,E2 -11933.562} C_VEL
LIN {X 0,Y 385.566,Z 405.363,A -85,B 0,C 180,E1 -11936.228,E2 -11936.228} C_VEL
LIN {X 0,Y 386.361,Z 411.149,A -85,B 0,C 180,E1 -11938.754,E2 -11938.754} C_VEL
LIN {X 0,Y 385.684,Z 416.881,A -85,B 0,C 180,E1 -11941.006,E2 -11941.006} C_VEL
LIN {X 0,Y 384.572,Z 426.206,A -85,B 0,C 180,E1 -11944.57,E2 -11944.57} C_VEL
LIN {X 0,Y 383.534,Z 436.995,A -85,B 0,C 180,E1 -11948.504,E2 -11948.504} C_VEL
LIN {X 0,Y 382.9,Z 445.366,A -85,B 0,C 180,E1 -11951.477,E2 -11951.477} C_VEL
LIN {X 0,Y 385.184,Z 458.806,A -85,B 0,C 180,E1 -11952.009,E2 -11952.009} C_VEL
LIN {X 0,Y 386.363,Z 469.883,A -85,B 0,C 180,E1 -11952.596,E2 -11952.596} C_VEL
LIN {X 0,Y 386.764,Z 477.681,A -85,B 0,C 180,E1 -11953.101,E2 -11953.101} C_VEL
LIN {X 0,Y 385.86,Z 489.822,A -85,B 0,C 180,E1 -11954.012,E2 -11954.012} C_VEL
LIN {X 0,Y 384.914,Z 500.557,A -85,B 0,C 180,E1 -11955.057,E2 -11955.057} C_VEL
LIN {X 0,Y 384.131,Z 510.31,A -85,B 0,C 180,E1 -11956.243,E2 -11956.243} C_VEL
LIN {X 0,Y 383.446,Z 519.151,A -85,B 0,C 180,E1 -11957.566,E2 -11957.566} C_VEL
LIN {X 0,Y 382.653,Z 528.103,A -85,B 0,C 180,E1 -11959.152,E2 -11959.152} C_VEL
LIN {X 0,Y 382.186,Z 535.385,A -85,B 0,C 180,E1 -11960.743,E2 -11960.743} C_VEL
LIN {X 0,Y 381.915,Z 540.278,A -85,B 0,C 180,E1 -11962.07,E2 -11962.07} C_VEL
LIN {X 0,Y 381.638,Z 545.741,A -85,B 0,C 180,E1 -11963.953,E2 -11963.953} C_VEL
LIN {X 0,Y 381.644,Z 549.513,A -85,B 0,C 180,E1 -11965.778,E2 -11965.778} C_VEL
LIN {X 0,Y 381.574,Z 551.094,A -85,B 0,C 180,E1 -11966.835,E2 -11966.835} C_VEL
LIN {X 0,Y 381.635,Z 552.237,A -85,B 0,C 180,E1 -11967.892,E2 -11967.892} C_VEL
